(*
==============================================================================
 Method: EstimateTotalTime
------------------------------------------------------------------------------
 Purpose:
   - Estimate the total duration (in seconds) of the prime phase for the
     current recipe, based on how many different solvents (1..4) are used.
   - This is used solely for the HMI progress bar to give a rough visual
     indication of progress.

 Logic:
   1) Build a local array bLocalPrimeRequired[1..4] from the recipe, similar
      to BuildPrimeListFromRecipe.
   2) Count how many solvents are required (iCount).
   3) If iCount = 0 → return a small non-zero time (1.0 s) to avoid div by 0.
   4) Else → estimate = rTimePerSolvent * iCount * 7
      (the factor 7 is an empirical scaling based on test runs).
==============================================================================
*)
METHOD EstimateTotalTime : REAL
VAR
    iStage              : INT;
    iSolventNum         : INT;
    bLocalPrimeRequired : ARRAY[1..4] OF BOOL := [FALSE, FALSE, FALSE, FALSE];
    iCount              : INT := 0;
    rTimePerSolvent     : REAL := 15.0;   // Approximate time (s) to prime one solvent
END_VAR
// Build a local "prime required" list based on the active recipe
FOR iStage := 1 TO 4 DO
    iSolventNum := GVL_Recipe.stActiveRecipe.stSolventsTimes.aSolventN[iStage];

    IF (iSolventNum >= 1) AND (iSolventNum <= 4) THEN
        bLocalPrimeRequired[iSolventNum] := TRUE;
    END_IF
END_FOR

// Count how many solvents need priming
FOR iStage := 1 TO 4 DO
    IF bLocalPrimeRequired[iStage] THEN
        iCount := iCount + 1;
    END_IF
END_FOR

// If nothing to prime, return a small value to avoid division by zero
IF iCount = 0 THEN
    EstimateTotalTime := 1.0;
ELSE
    EstimateTotalTime := rTimePerSolvent * TO_REAL(iCount) * 7.0;
END_IF
END_METHOD

ACTION PrimeSolventCycle:
(*
==============================================================================
 PrimeSolventCycle
------------------------------------------------------------------------------
 Purpose:
   - Execute the generic prime cycle for the solvent indicated by
     iActiveSolventPosition (1..4).
   - This action uses iStepCounter as an internal step machine and sets
     bMovementComplete := TRUE when the cycle for the current solvent
     is finished.

 Prime sequence (per solvent):
   0) Initialise flags and HMI text for current solvent.
   1) Set valves [1..5] to the solvent position (1..4).
   2) Compute pump forward distances for rPrimeForwardVolume (ml).
   3) Pump forward (positive Distance) to pull solvent from bottle
      through the lines and into jars.
   4) Set valves [1..5] to needles position (6).
   5) Compute pump backward distances for rPrimeBackwardVolume (ml).
   6) Pump backward (negative Distance) to empty jars while keeping
      the lines filled with solvent.
   7) Set bMovementComplete := TRUE (cycle finished).
==============================================================================
*)

CASE iStepCounter OF

    // -------------------------------------------------------------
    // 0) Initialise HMI state and clear flags
    // -------------------------------------------------------------
    0:
        CASE iActiveSolventPosition OF
            1: GVL_HMI.HMIAnimation.sLoadTextRecovery := 'Prime Solvent 1';
            2: GVL_HMI.HMIAnimation.sLoadTextRecovery := 'Prime Solvent 2';
            3: GVL_HMI.HMIAnimation.sLoadTextRecovery := 'Prime Solvent 3';
            4: GVL_HMI.HMIAnimation.sLoadTextRecovery := 'Prime Solvent 4';
        ELSE
            GVL_HMI.HMIAnimation.sLoadTextRecovery := 'Prime Solvent';
        END_CASE;

        // Reset valve flags
        FOR i := 1 TO 5 DO
            bMoveValveDone[i] := FALSE;
        END_FOR

        // Reset pump flags and distances
        FOR i := 1 TO 10 DO
            bMovePumpDone[i] := FALSE;
            fDistance[i]     := 0.0;
        END_FOR

        bMovementComplete := FALSE;
        iStepCounter      := 1;


    // -------------------------------------------------------------
    // 1) Set valves [1..5] to the solvent position (1..4)
    // -------------------------------------------------------------
    1:
        FOR i := 1 TO 5 DO
            IF NOT bMoveValveDone[i] THEN
                bMoveValveDone[i] := GVL_Motion.aValvesObj[i].MoveValve(
                    iPosition := iActiveSolventPosition,   // solvent position 1..4
                    rVelocity := GVL_Motion.aValves[i].rTargetVel,
                    rAcc      := GVL_Motion.aValves[i].rAcceleration,
                    rDec      := GVL_Motion.aValves[i].rDeceleration
                );
            END_IF
        END_FOR

        // Wait until all valves reach solvent position
        IF bMoveValveDone[1] AND bMoveValveDone[2] AND bMoveValveDone[3]
           AND bMoveValveDone[4] AND bMoveValveDone[5] THEN

            FOR i := 1 TO 5 DO
                bMoveValveDone[i] := FALSE;
            END_FOR

            iStepCounter := 2;
        END_IF


    // -------------------------------------------------------------
    // 2) Calculate forward distance for rPrimeForwardVolume
    // -------------------------------------------------------------
    2:
        FOR i := 1 TO 10 DO
            fDistance[i] := F_VolumeToSteps(
                rVolume    := rPrimeForwardVolume,   // Forward prime volume
                iPumpIndex := i
            );
            bMovePumpDone[i] := FALSE;
        END_FOR

        iStepCounter := 3;


    // -------------------------------------------------------------
    // 3) Pump forward (positive movement) to fill lines and jars
    // -------------------------------------------------------------
    3:
        FOR i := 1 TO 10 DO
            IF NOT bMovePumpDone[i] THEN
                bMovePumpDone[i] := GVL_Motion.aPumpsRotary[i].MoveRelative(
                    Distance := fDistance[i],  // positive → forward
                    Velocity := GVL_Settings.stPumpParameters.iMeterVelocity * 6,
                    Acc      := GVL_Settings.stPumpParameters.iMeterVelocity * 3,
                    Dec      := GVL_Settings.stPumpParameters.iMeterVelocity * 3
                );
            END_IF
        END_FOR

        // Wait until all pumps finish forward prime
        IF bMovePumpDone[1] AND bMovePumpDone[2] AND bMovePumpDone[3] AND
           bMovePumpDone[4] AND bMovePumpDone[5] AND bMovePumpDone[6] AND
           bMovePumpDone[7] AND bMovePumpDone[8] AND bMovePumpDone[9] AND
           bMovePumpDone[10] THEN

            FOR i := 1 TO 10 DO
                bMovePumpDone[i] := FALSE;
            END_FOR

            iStepCounter := 4;
        END_IF


    // -------------------------------------------------------------
    // 4) Set valves [1..5] to needles position (6)
    // -------------------------------------------------------------
    4:
        FOR i := 1 TO 5 DO
            IF NOT bMoveValveDone[i] THEN
                bMoveValveDone[i] := GVL_Motion.aValvesObj[i].MoveValve(
                    iPosition := 6,   // needles position
                    rVelocity := GVL_Motion.aValves[i].rTargetVel,
                    rAcc      := GVL_Motion.aValves[i].rAcceleration,
                    rDec      := GVL_Motion.aValves[i].rDeceleration
                );
            END_IF
        END_FOR

        // Wait until all valves are at needles position
        IF bMoveValveDone[1] AND bMoveValveDone[2] AND bMoveValveDone[3]
           AND bMoveValveDone[4] AND bMoveValveDone[5] THEN

            FOR i := 1 TO 5 DO
                bMoveValveDone[i] := FALSE;
            END_FOR

            iStepCounter := 5;
        END_IF


    // -------------------------------------------------------------
    // 5) Calculate backward distance for rPrimeBackwardVolume
    // -------------------------------------------------------------
    5:
        FOR i := 1 TO 10 DO
            fDistance[i] := F_VolumeToSteps(
                rVolume    := rPrimeBackwardVolume,  // Backward prime volume
                iPumpIndex := i
            );
            bMovePumpDone[i] := FALSE;
        END_FOR

        iStepCounter := 6;


    // -------------------------------------------------------------
    // 6) Pump backward (negative movement) to empty jars into waste
    // -------------------------------------------------------------
    6:
        FOR i := 1 TO 10 DO
            IF NOT bMovePumpDone[i] THEN
                bMovePumpDone[i] := GVL_Motion.aPumpsRotary[i].MoveRelative(
                    Distance := -fDistance[i],  // negative → backward
                    Velocity := GVL_Settings.stPumpParameters.iRunVelocity * 6,
                    Acc      := GVL_Settings.stPumpParameters.iRunVelocity * 3,
                    Dec      := GVL_Settings.stPumpParameters.iRunVelocity * 3
                );
            END_IF
        END_FOR

        // Wait until all pumps finish backward cycle
        IF bMovePumpDone[1] AND bMovePumpDone[2] AND bMovePumpDone[3] AND
           bMovePumpDone[4] AND bMovePumpDone[5] AND bMovePumpDone[6] AND
           bMovePumpDone[7] AND bMovePumpDone[8] AND bMovePumpDone[9] AND
           bMovePumpDone[10] THEN

            FOR i := 1 TO 10 DO
                bMovePumpDone[i] := FALSE;
            END_FOR

            iStepCounter := 7;
        END_IF


    // -------------------------------------------------------------
    // 7) Prime cycle finished for this solvent
    // -------------------------------------------------------------
    7:
        bMovementComplete := TRUE;

END_CASE
END_ACTION

(*
==============================================================================
 Method: Reset
------------------------------------------------------------------------------
 Purpose:
   - Reset all internal flags, counters, and HMI fields associated with the
     prime phase, so that a new prime sequence can start cleanly.

 Behaviour:
   - Clears:
       * bStart, bBusy, bDone, bError, bProgressInitDone
       * ePrimeState, iStepCounter, bMovementComplete
       * bMoveValveDone[], bMovePumpDone[], fDistance[]
       * HMI prime text / bar (Recovery text cleared here as well)
   - Returns:
       Reset = TRUE once the operation is completed.
==============================================================================
*)
METHOD Reset : BOOL
VAR
    j : INT;
END_VAR
Reset := FALSE;

// Clear basic state and flags
bStart            := FALSE;
bBusy             := FALSE;
bDone             := FALSE;
bError            := FALSE;
bProgressInitDone := FALSE;

ePrimeState       := E_PrimeSolventState.PS_Idle;
iStepCounter      := 0;
bMovementComplete := FALSE;

// Clear motion flags and distances
FOR j := 1 TO 5 DO
    bMoveValveDone[j] := FALSE;
END_FOR

FOR j := 1 TO 10 DO
    bMovePumpDone[j] := FALSE;
    fDistance[j]     := 0.0;
END_FOR

// Clear HMI texts for prime / recovery bars if needed
GVL_HMI.HMIAnimation.sLoadTextRecovery := '';
GVL_HMI.HMIAnimation.rLoadBarRecovery  := 0.0;

// Mark reset as completed
Reset := TRUE;
RETURN;
END_METHOD

END_FUNCTION_BLOCK

// ---- POUs/Functions/F_AnyAxisMoving.TcPOU
FUNCTION F_AnyAxisMoving : BOOL
VAR_INPUT
END_VAR
VAR
	i : INT;
END_VAR

F_AnyAxisMoving := FALSE;

// Motors M1 - M3

F_AnyAxisMoving := F_AnyAxisMoving  OR (NOT GVL_Motion.M1Motor.iNotMoving)
									OR (NOT GVL_Motion.M2Motor.iNotMoving)
									OR (NOT GVL_Motion.M3Motor.iNotMoving);

// VICI Valves
FOR i := 1 TO 5 DO
    F_AnyAxisMoving := F_AnyAxisMoving 
        OR (NOT GVL_Motion.aValves[i].iNotMoving);
END_FOR

// Linear pumps
FOR i := 1 TO 10 DO
    F_AnyAxisMoving := F_AnyAxisMoving 
        OR (NOT GVL_Motion.aPumps[i].Linear.iNotMoving);
END_FOR

// Rotary pumps
FOR i := 1 TO 10 DO
    F_AnyAxisMoving := F_AnyAxisMoving 
        OR (NOT GVL_Motion.aPumps[i].Rotary.iNotMoving);
END_FOR

END_FUNCTION

// ---- POUs/1. MachineControl/PRG_SystemInit.TcPOU
PROGRAM PRG_SystemInit
VAR_OUTPUT
	bDone           : BOOL := FALSE;
END_VAR
VAR
	i               : INT;
	j				: INT;
    bAllDone        : BOOL := FALSE;
    bStartedAction  : BOOL := FALSE;
	bMoveZeroDone	: BOOL := FALSE;
    bInitComplete   : BOOL := FALSE;
	bVerticalMotorsDone		: BOOL := FALSE;   
	bLinearMotorsHomingDone	: BOOL := FALSE; 
	bValvesHomingDone 		: BOOL := FALSE;
	bLinearPumpsDone		: BOOL := FALSE;
	bPerformHoming			: BOOL := FALSE;
	
	bAllResetDone		: BOOL := FALSE;
	bEnableDone			: BOOL := FALSE;
	bResetCheck			: ARRAY[1..28] OF BOOL;
	
	aMotorsEnabled 	: ARRAY[1..3] OF BOOL;
	aValvesEnabled 	: ARRAY[1..5] OF BOOL;
	aLinearPumpsEnabled	: ARRAY[1..10] OF BOOL;
	aRotaryPumpsEnabled	: ARRAY[1..10] OF BOOL;
	
	bAllPumpsEnabled  : BOOL := FALSE;
	bAllLinearPumpsEnabled  : BOOL := FALSE;
	bAllRotaryPumpsEnabled  : BOOL := FALSE;
	bAllMotorsEnabled : BOOL := FALSE;
	bAllValvesEnabled : BOOL := FALSE;
	
	bHomeMotorDone	: ARRAY[1..3] OF BOOL;
	bHomeValveDone  : ARRAY[1..5] OF BOOL;
	bHomePumpDone	: ARRAY[1..10] OF BOOL;
	
	bM2InPosition	: BOOL;
	rPosTolerance	: REAL := 1.0;
	
	bMoveValve1Request	: BOOL := TRUE;
	bMoveValve2Request	: BOOL := TRUE;
	
	bMoveMotorsRequest	: ARRAY[1..3] OF BOOL;
	bMoveMotorDone		: ARRAY[1..3] OF BOOL;
	
	bCalibrationReset	  : BOOL := FALSE;
	bManualModeReset	  : BOOL := FALSE;
	bAutoCycleReset		  : BOOL := FALSE;
	bAllLogicResetDone	  : BOOL := FALSE;
	bInitLogicLatchesDone : BOOL := FALSE;
	
	tonResetDelay	: ton;
	tonEnableDelay	: ton;
	
	//Timeout timers for each step
	tonResetTimeOut		: ton;
	tonEnableTimeOut	: ton;
	tonHomeTimeOut		: ton;
	tonMoveAbsTimeOut	: ton;
		
	stStatus : ST_ActuatorStatus;
	
END_VAR

// ============================================================================
// PRG_SystemInit
// Handles full system initialization sequence:
//  0) Reset PRG's Manual | Calibration | AutoCycle
//  1) Reset all axes (motors, valves, pumps)
//  2) Enable all required axes
//  3) Perform homing on first startup OR move axes to zero on subsequent inits
//  4) Check completion and errors
//  5) Set bDone when initialization is complete
// ============================================================================

// ---------------------------------------------------------------------------
// 0) Basic delays between phases
// ---------------------------------------------------------------------------

// Delay before starting Reset
tonResetDelay(
    IN := NOT bAllResetDone,
    PT := T#1S
);

// Delay before starting Enable (only after Reset is fully done)
tonEnableDelay(
    IN := bAllResetDone AND NOT bEnableDone,
    PT := T#1S
);

// ---------------------------------------------------------------------------
// 0) Step 0 - Reset all logic Flags, PRGs and FBs
// ---------------------------------------------------------------------------
IF NOT bInitLogicLatchesDone AND GVL_Motion.bValvesPositionRecovered THEN ACT_ResetCommandFlags(); END_IF // Valves position recovery after shutdown change | Renan 22Jan2026

IF NOT bAllLogicResetDone AND bInitLogicLatchesDone THEN ACT_LogicResets(); END_IF

// ---------------------------------------------------------------------------
// 1) Step 1 - Reset all axes (motors, valves, linear and rotary pumps)
// ---------------------------------------------------------------------------
IF NOT bAllResetDone AND bAllLogicResetDone AND bInitLogicLatchesDone AND tonResetDelay.Q THEN
    ACT_ResetMotors();   // Uses bResetCheck[1..28], tonResetTimeOut, etc.
END_IF

// ---------------------------------------------------------------------------
// 2) Step 2 - Enable all axes (motors, valves, rotary pumps)
//     - Uses extra layer: checks Axis.Status.Error before/after Enable
// ---------------------------------------------------------------------------
IF bAllResetDone AND NOT bEnableDone AND tonEnableDelay.Q THEN
    ACT_EnableMotors();
END_IF

// ---------------------------------------------------------------------------
// 3) Step 3 - Decide if we need Homing or only MoveToZero
//     - First SystemInit: perform homing (bInitialHomingDone = FALSE)
//     - Next SystemInits: only move motors/valves to zero/home position
// ---------------------------------------------------------------------------

IF NOT bStartedAction AND bAllResetDone AND bEnableDone THEN
    bStartedAction := TRUE;

    // First time the machine starts: perform initial homing
    IF NOT GVL_Motion.bInitialHomingDone THEN
        bPerformHoming := TRUE;   // ACT_Homing() will be called
    ELSE
        bPerformHoming := FALSE;  // ACT_MoveToZero() will be called
    END_IF
END_IF

// ---------------------------------------------------------------------------
// 3a) Execute Homing or MoveToZero depending on bPerformHoming
// ---------------------------------------------------------------------------
IF bStartedAction THEN
    IF bPerformHoming THEN
        ACT_Homing();
    ELSE
        ACT_MoveToZero();
    END_IF
END_IF

// ---------------------------------------------------------------------------
// 4) Step 4 + 5 - Check if all motors and valves have completed their action
//     - Also checks for errors from wrapper (stStatus.bError)
//       and directly from Axis.Status.Error
// ---------------------------------------------------------------------------
IF bStartedAction AND bMoveZeroDone THEN
    bAllDone := TRUE;

    // Check motors M1..M3
    FOR i := 1 TO 3 DO
        stStatus := GVL_Motion.aMotors[i].GetStatus();

        // If any motor is not done yet
        IF NOT stStatus.bDone THEN
            bAllDone := FALSE;
        END_IF

        // If any motor returned an error (wrapper OR Axis), abort with immediate fault
        IF stStatus.bError THEN
            GVL_HMI.eMachineMode := E_MachineMode.IMEDIATE_FAULT;
            RETURN;
        END_IF
    END_FOR

    // Check valves V1..V5
    FOR i := 1 TO 5 DO
        stStatus := GVL_Motion.aValvesObj[i].GetStatus();

        // If any valve is not done yet
        IF NOT stStatus.bDone THEN
            bAllDone := FALSE;
        END_IF

        // If any valve returned an error (wrapper OR Axis), abort with immediate fault
        IF stStatus.bError THEN
            GVL_HMI.eMachineMode := E_MachineMode.IMEDIATE_FAULT;
            RETURN;
        END_IF
    END_FOR
END_IF

// ---------------------------------------------------------------------------
// 5) Step 6 - Finalization of System Init
//     - Set bDone only when Reset, Enable and Actions are all completed
// ---------------------------------------------------------------------------
IF bAllDone AND bAllResetDone AND bEnableDone AND NOT bInitComplete THEN
    bInitComplete := TRUE;
    bDone         := TRUE;

    // Mark that the initial homing has been successfully completed
    IF NOT GVL_Motion.bInitialHomingDone THEN
        GVL_Motion.bInitialHomingDone := TRUE;
    END_IF
END_IF

ACTION ACT_EnableMotors:
// ============================================================================
// Step 2: Enable all motors, valves and rotary pumps
//   - Uses aMotorsEnabled[1..3], aValvesEnabled[1..5], aRotaryPumpsEnabled[1..10]
//   - Sets bAllMotorsEnabled, bAllValvesEnabled, bAllRotaryPumpsEnabled
//   - Uses tonEnableTimeOut and GVL_Alarms.sMotionEnableTimeoutAxis
//   - Extra layer: checks wrapper error (GetStatus().bError) before enabling
// ============================================================================

IF NOT bEnableDone THEN

    // Assume all will be enabled, then AND with each device
    bAllMotorsEnabled      := TRUE;
    bAllValvesEnabled      := TRUE;
    bAllRotaryPumpsEnabled := TRUE;

    // -----------------------------
    // 2.1 Motors (M1..M3)
    // -----------------------------
    FOR i := 1 TO 3 DO
        // Read wrapper status
        stStatus := GVL_Motion.aMotors[i].GetStatus();

        // If wrapper reports error at this stage, abort System Init
        IF stStatus.bError THEN
            GVL_HMI.eMachineMode := E_MachineMode.IMEDIATE_FAULT;
            RETURN;
        END_IF

        // If axis is disabled, request Enable through wrapper
        // (If your wrapper has a specific bEnabled flag, you can check it here.
        // Otherwise, just call Enable() and rely on the wrapper to handle it.)
        aMotorsEnabled[i] := GVL_Motion.aMotors[i].Enable();

        bAllMotorsEnabled := bAllMotorsEnabled AND aMotorsEnabled[i];
    END_FOR

    // -----------------------------
    // 2.2 Valves (V1..V5)
    // -----------------------------
    FOR i := 1 TO 5 DO
        stStatus := GVL_Motion.aValvesObj[i].GetStatus();

        IF stStatus.bError THEN
            GVL_HMI.eMachineMode := E_MachineMode.IMEDIATE_FAULT;
            RETURN;
        END_IF

        aValvesEnabled[i] := GVL_Motion.aValvesObj[i].Enable();

        bAllValvesEnabled := bAllValvesEnabled AND aValvesEnabled[i];
    END_FOR

    // -----------------------------
    // 2.3 Rotary pumps (RP1..RP10)
// -----------------------------
    FOR i := 1 TO 10 DO
        stStatus := GVL_Motion.aPumpsRotary[i].GetStatus();

        IF stStatus.bError THEN
            GVL_HMI.eMachineMode := E_MachineMode.IMEDIATE_FAULT;
            RETURN;
        END_IF

        aRotaryPumpsEnabled[i] := GVL_Motion.aPumpsRotary[i].Enable();

        bAllRotaryPumpsEnabled := bAllRotaryPumpsEnabled AND aRotaryPumpsEnabled[i];
    END_FOR

    // -----------------------------
    // 2.4 Enable timeout monitoring and alarm
    // -----------------------------
    tonEnableTimeOut(IN := TRUE, PT := T#10S);

    IF tonEnableTimeOut.Q AND NOT (bAllMotorsEnabled AND bAllValvesEnabled AND bAllRotaryPumpsEnabled) THEN
        // Build string with axes that were NOT enabled within timeout

        // Motors M1..M3
        FOR i := 1 TO 3 DO
            IF NOT aMotorsEnabled[i] THEN
                IF GVL_Alarms.sMotionEnableTimeoutAxis <> '' THEN
                    GVL_Alarms.sMotionEnableTimeoutAxis :=
                        CONCAT(GVL_Alarms.sMotionEnableTimeoutAxis, ', ');
                END_IF
                GVL_Alarms.sMotionEnableTimeoutAxis :=
                    CONCAT(GVL_Alarms.sMotionEnableTimeoutAxis,
                           GVL_Constant.sMotionText[i]);
            END_IF
        END_FOR

        // Valves V1..V5
        FOR i := 1 TO 5 DO
            IF NOT aValvesEnabled[i] THEN
                IF GVL_Alarms.sMotionEnableTimeoutAxis <> '' THEN
                    GVL_Alarms.sMotionEnableTimeoutAxis :=
                        CONCAT(GVL_Alarms.sMotionEnableTimeoutAxis, ', ');
                END_IF
                GVL_Alarms.sMotionEnableTimeoutAxis :=
                    CONCAT(GVL_Alarms.sMotionEnableTimeoutAxis,
                           GVL_Constant.sMotionText[i + 3]);
            END_IF
        END_FOR

        // Rotary pumps RP1..RP10
        FOR i := 1 TO 10 DO
            IF NOT aRotaryPumpsEnabled[i] THEN
                IF GVL_Alarms.sMotionEnableTimeoutAxis <> '' THEN
                    GVL_Alarms.sMotionEnableTimeoutAxis :=
                        CONCAT(GVL_Alarms.sMotionEnableTimeoutAxis, ', ');
                END_IF
                GVL_Alarms.sMotionEnableTimeoutAxis :=
                    CONCAT(GVL_Alarms.sMotionEnableTimeoutAxis,
                           GVL_Constant.sMotionText[i + 18]);
            END_IF
        END_FOR

        GVL_Alarms.bMotionEnableTimeout := TRUE;
        // Strong robustness: abort System Init on enable timeout
        GVL_HMI.eMachineMode := E_MachineMode.IMEDIATE_FAULT;
        RETURN;
    END_IF

    // -----------------------------
    // 2.5 Step completion
    // -----------------------------
    IF bAllMotorsEnabled AND bAllValvesEnabled AND bAllRotaryPumpsEnabled THEN
        bEnableDone := TRUE;
        tonEnableTimeOut(IN := FALSE);
    END_IF

ELSE
    // Already done, ensure timer is off
    tonEnableTimeOut(IN := FALSE);
END_IF
END_ACTION

ACTION ACT_Homing:
// ============================================================================
// Step 3 (part 1): Initial homing sequence
//   - Only used when GVL_Motion.bInitialHomingDone = FALSE
//   - Homes vertical motors, then horizontal motor
//   - Moves valves to home position (position 5) when positions are recovered
//   - Monitors homing timeout and raises alarm
// ============================================================================

IF bPerformHoming THEN

    // -----------------------------
    // 3.1 Vertical motors homing (M1, M2)
    // -----------------------------
    IF NOT bHomeMotorDone[1] THEN
        bHomeMotorDone[1] := GVL_Motion.aMotors[1].Home(
            pHomeSensor := ADR(GVL_IO.gDigInputs.bStageCollection_Home),
            rVelocity   := GVL_Motion.M1Motor.rHomeVel,
            rAcc        := GVL_Motion.M1Motor.rHomeAcc,
            rDec        := GVL_Motion.M1Motor.rHomeDec
        );
    END_IF

    IF NOT bHomeMotorDone[2] THEN
        bHomeMotorDone[2] := GVL_Motion.aMotors[2].Home(
            pHomeSensor := ADR(GVL_IO.gDigInputs.bSampleRecovery_Vertical_Home),
            rVelocity   := GVL_Motion.M2Motor.rHomeVel,
            rAcc        := GVL_Motion.M2Motor.rHomeAcc,
            rDec        := GVL_Motion.M2Motor.rHomeDec
        );
    END_IF

    // Check if vertical motors homing is done
    IF bHomeMotorDone[1] AND bHomeMotorDone[2] THEN
        bVerticalMotorsDone := TRUE;
    END_IF

    // -----------------------------
    // 3.2 Horizontal motor homing (M3), only after verticals are done
    // -----------------------------
    IF bVerticalMotorsDone AND NOT bHomeMotorDone[3] THEN
        bHomeMotorDone[3] := GVL_Motion.aMotors[3].Home(
            pHomeSensor := ADR(GVL_IO.gDigInputs.bSampleRecovery_Horizontal_Home),
            rVelocity   := GVL_Motion.M3Motor.rHomeVel,
            rAcc        := GVL_Motion.M3Motor.rHomeAcc,
            rDec        := GVL_Motion.M3Motor.rHomeDec
        );
    END_IF

    // Check if all linear motors are homed
    IF bHomeMotorDone[1] AND bHomeMotorDone[2] AND bHomeMotorDone[3] THEN
        bLinearMotorsHomingDone := TRUE;
    END_IF

    // -----------------------------
    // 3.3 Valves homing (move to position 5) if position is recovered
    // -----------------------------
    IF GVL_Motion.bValvesPositionRecovered THEN
        // Move all valves to position 5 (home position)
        IF NOT bHomeValveDone[1] THEN
            bHomeValveDone[1] := GVL_Motion.aValvesObj[1].MoveValve(
                iPosition := 5,
                rVelocity := GVL_Motion.aValves[1].rHomeVel,
                rAcc      := GVL_Motion.aValves[1].rHomeAcc,
                rDec      := GVL_Motion.aValves[1].rHomeDec
            );
        END_IF

        IF NOT bHomeValveDone[2] THEN
            bHomeValveDone[2] := GVL_Motion.aValvesObj[2].MoveValve(
                iPosition := 5,
                rVelocity := GVL_Motion.aValves[2].rHomeVel,
                rAcc      := GVL_Motion.aValves[2].rHomeAcc,
                rDec      := GVL_Motion.aValves[2].rHomeDec
            );
        END_IF

        IF NOT bHomeValveDone[3] THEN
            bHomeValveDone[3] := GVL_Motion.aValvesObj[3].MoveValve(
                iPosition := 5,
                rVelocity := GVL_Motion.aValves[3].rHomeVel,
                rAcc      := GVL_Motion.aValves[3].rHomeAcc,
                rDec      := GVL_Motion.aValves[3].rHomeDec
            );
        END_IF

        IF NOT bHomeValveDone[4] THEN
            bHomeValveDone[4] := GVL_Motion.aValvesObj[4].MoveValve(
                iPosition := 5,
                rVelocity := GVL_Motion.aValves[4].rHomeVel,
                rAcc      := GVL_Motion.aValves[4].rHomeAcc,
                rDec      := GVL_Motion.aValves[4].rHomeDec
            );
        END_IF

        IF NOT bHomeValveDone[5] THEN
            bHomeValveDone[5] := GVL_Motion.aValvesObj[5].MoveValve(
                iPosition := 5,
                rVelocity := GVL_Motion.aValves[5].rHomeVel,
                rAcc      := GVL_Motion.aValves[5].rHomeAcc,
                rDec      := GVL_Motion.aValves[5].rHomeDec
            );
        END_IF
    END_IF

    // Check if all valves homing are done
    bValvesHomingDone :=
        bHomeValveDone[1] AND bHomeValveDone[2] AND bHomeValveDone[3] AND
        bHomeValveDone[4] AND bHomeValveDone[5];

	// If all motors and valves completed their homing, finalize
	IF bLinearMotorsHomingDone AND bValvesHomingDone THEN 
		bMoveZeroDone := TRUE;
	END_IF	
	
    // -----------------------------
    // 3.4 Homing timeout monitoring and alarm
    // -----------------------------
    tonHomeTimeOut(
        IN := NOT (bLinearMotorsHomingDone AND bValvesHomingDone),
        PT := T#40S
    );

    IF tonHomeTimeOut.Q AND NOT (bLinearMotorsHomingDone AND bValvesHomingDone) THEN
        // Build string with axes that were NOT homed in time

        // Motors M1..M3
        FOR j := 1 TO 3 DO
            IF NOT bHomeMotorDone[j] THEN
                IF GVL_Alarms.sMotionHomeTimeoutAxis <> '' THEN
                    GVL_Alarms.sMotionHomeTimeoutAxis :=
                        CONCAT(GVL_Alarms.sMotionHomeTimeoutAxis, ', ');
                END_IF
                GVL_Alarms.sMotionHomeTimeoutAxis :=
                    CONCAT(GVL_Alarms.sMotionHomeTimeoutAxis,
                           GVL_Constant.sMotionText[j]);
            END_IF
        END_FOR

        // Valves V1..V5
        FOR j := 1 TO 5 DO
            IF NOT bHomeValveDone[j] THEN
                IF GVL_Alarms.sMotionHomeTimeoutAxis <> '' THEN
                    GVL_Alarms.sMotionHomeTimeoutAxis :=
                        CONCAT(GVL_Alarms.sMotionHomeTimeoutAxis, ', ');
                END_IF
                GVL_Alarms.sMotionHomeTimeoutAxis :=
                    CONCAT(GVL_Alarms.sMotionHomeTimeoutAxis,
                           GVL_Constant.sMotionText[j + 3]);
            END_IF
        END_FOR

        GVL_Alarms.bMotionHomeTimeout := TRUE;
        GVL_HMI.eMachineMode          := E_MachineMode.IMEDIATE_FAULT;
    END_IF

END_IF
END_ACTION

ACTION ACT_LogicResets:
IF NOT bAllLogicResetDone THEN
	
	bCalibrationReset	:= PRG_Calibration.Reset();
	bManualModeReset	:= PRG_ManualControl.Reset();
	bAutoCycleReset		:= PRG_AutoCycle.Reset();
	
	IF bCalibrationReset AND bManualModeReset AND bAutoCycleReset THEN
		bAllLogicResetDone 	:= TRUE;
	END_IF
	
END_IF
END_ACTION

ACTION ACT_MoveToZero:
// ============================================================================
// Step 3 (part 2): Move motors and valves to zero / default positions
//   - Used when GVL_Motion.bInitialHomingDone = TRUE
//   - Moves:
//       - M1, M2, M3 -> position 0.0
//       - Valves V1..V5 -> position 5
//   - Uses bMoveMotorDone[1..3] and bHomeValveDone[1..5]
//   - Monitors move absolute timeout and raises alarm
// ============================================================================

IF NOT bPerformHoming THEN

    // -----------------------------
    // 3.5 Move linear motors to 0.0
    // -----------------------------
    // You can adjust these velocity/acc/dec parameters as needed
    IF NOT bMoveMotorDone[1] THEN
        bMoveMotorDone[1] := GVL_Motion.aMotors[1].MoveAbsolute(
            rPosition := GVL_Settings.stMachineParam.aM1Position[1],
            rVelocity := GVL_Settings.stMachineParam.rM1Velocity,
            rAcc      := GVL_Settings.stMachineParam.rM1Accleration,
            rDec      := GVL_Settings.stMachineParam.rM1Deceleration
        );
    END_IF

    IF NOT bMoveMotorDone[2] THEN
        bMoveMotorDone[2] := GVL_Motion.aMotors[2].MoveAbsolute(
            rPosition := GVL_Settings.stMachineParam.aM2Position[1],
            rVelocity := GVL_Settings.stMachineParam.rM2Velocity,
            rAcc      := GVL_Settings.stMachineParam.rM2Accleration,
            rDec      := GVL_Settings.stMachineParam.rM2Deceleration
        );
    END_IF
	
	// Track real M2 Position before start moving M3 
	bM2InPosition := ABS(GVL_Motion.M2Motor.rActualPos - GVL_Settings.stMachineParam.aM2Position[1]) < rPosTolerance;
	
    IF bMoveMotorDone[2] AND bM2InPosition AND NOT bMoveMotorDone[3] THEN
        bMoveMotorDone[3] := GVL_Motion.aMotors[3].MoveAbsolute(
            rPosition := GVL_Settings.stMachineParam.aM3Position[1],
            rVelocity := GVL_Settings.stMachineParam.rM3Velocity,
            rAcc      := GVL_Settings.stMachineParam.rM3Accleration,
            rDec      := GVL_Settings.stMachineParam.rM3Deceleration
        );
    END_IF

    // Linear motors move done flag
    bLinearMotorsHomingDone :=
        bMoveMotorDone[1] AND bMoveMotorDone[2] AND bMoveMotorDone[3];

    // -----------------------------
    // 3.6 Move valves to position 5 (default/home position)
// -----------------------------
    IF NOT bHomeValveDone[1] THEN
        bHomeValveDone[1] := GVL_Motion.aValvesObj[1].MoveValve(
            iPosition := 5,
            rVelocity := GVL_Motion.aValves[1].rHomeVel,
            rAcc      := GVL_Motion.aValves[1].rHomeAcc,
            rDec      := GVL_Motion.aValves[1].rHomeDec
        );
    END_IF

    IF NOT bHomeValveDone[2] THEN
        bHomeValveDone[2] := GVL_Motion.aValvesObj[2].MoveValve(
            iPosition := 5,
            rVelocity := GVL_Motion.aValves[2].rHomeVel,
            rAcc      := GVL_Motion.aValves[2].rHomeAcc,
            rDec      := GVL_Motion.aValves[2].rHomeDec
        );
    END_IF

    IF NOT bHomeValveDone[3] THEN
        bHomeValveDone[3] := GVL_Motion.aValvesObj[3].MoveValve(
            iPosition := 5,
            rVelocity := GVL_Motion.aValves[3].rHomeVel,
            rAcc      := GVL_Motion.aValves[3].rHomeAcc,
            rDec      := GVL_Motion.aValves[3].rHomeDec
        );
    END_IF

    IF NOT bHomeValveDone[4] THEN
        bHomeValveDone[4] := GVL_Motion.aValvesObj[4].MoveValve(
            iPosition := 5,
            rVelocity := GVL_Motion.aValves[4].rHomeVel,
            rAcc      := GVL_Motion.aValves[4].rHomeAcc,
            rDec      := GVL_Motion.aValves[4].rHomeDec
        );
    END_IF

    IF NOT bHomeValveDone[5] THEN
        bHomeValveDone[5] := GVL_Motion.aValvesObj[5].MoveValve(
            iPosition := 5,
            rVelocity := GVL_Motion.aValves[5].rHomeVel,
            rAcc      := GVL_Motion.aValves[5].rHomeAcc,
            rDec      := GVL_Motion.aValves[5].rHomeDec
        );
    END_IF

    // Valves move done flag
    bValvesHomingDone :=
        bHomeValveDone[1] AND bHomeValveDone[2] AND
        bHomeValveDone[3] AND bHomeValveDone[4] AND bHomeValveDone[5];
	
	// If all motors and valves completed their homing, finalize
	IF bLinearMotorsHomingDone AND bValvesHomingDone THEN 
		bMoveZeroDone := TRUE;
	END_IF
	
    // -----------------------------
    // 3.7 MoveAbs timeout monitoring and alarm
    //    (Note: here we correctly use bMoveMotorDone instead of bHomeMotorDone)
// -----------------------------
    tonMoveAbsTimeOut(
        IN := NOT (bLinearMotorsHomingDone AND bValvesHomingDone),
        PT := T#40S
    );

    IF tonMoveAbsTimeOut.Q AND NOT (bLinearMotorsHomingDone AND bValvesHomingDone) THEN
        // Build string with axes that did NOT complete MoveAbsolute in time

        // Motors M1..M3
        FOR j := 1 TO 3 DO
            IF NOT bMoveMotorDone[j] THEN
                IF GVL_Alarms.sMotionMoveAbsTimeoutAxis <> '' THEN
                    GVL_Alarms.sMotionMoveAbsTimeoutAxis :=
                        CONCAT(GVL_Alarms.sMotionMoveAbsTimeoutAxis, ', ');
                END_IF
                GVL_Alarms.sMotionMoveAbsTimeoutAxis :=
                    CONCAT(GVL_Alarms.sMotionMoveAbsTimeoutAxis,
                           GVL_Constant.sMotionText[j]);
            END_IF
        END_FOR

        // Valves V1..V5
        FOR j := 1 TO 5 DO
            IF NOT bHomeValveDone[j] THEN
                IF GVL_Alarms.sMotionMoveAbsTimeoutAxis <> '' THEN
                    GVL_Alarms.sMotionMoveAbsTimeoutAxis :=
                        CONCAT(GVL_Alarms.sMotionMoveAbsTimeoutAxis, ', ');
                END_IF
                GVL_Alarms.sMotionMoveAbsTimeoutAxis :=
                    CONCAT(GVL_Alarms.sMotionMoveAbsTimeoutAxis,
                           GVL_Constant.sMotionText[j + 3]);
            END_IF
        END_FOR

        GVL_Alarms.bMotionMoveAbsTimeout := TRUE;
        GVL_HMI.eMachineMode             := E_MachineMode.IMEDIATE_FAULT;
    END_IF

END_IF
END_ACTION

ACTION ACT_ResetCommandFlags:
(*
    Action: ACT_ResetCommandFlags
    Purpose:
        Clear all HMI command flags and internal latched commands that might remain TRUE
        after an abnormal interruption (STOP/Abort), preventing unintended auto-start
        when re-entering a mode.

    Where to call:
        - PRG_StoppedState (first scan / when entering STOPPED)
        - PRG_SystemInit (first scan / at init start)

    Notes:
        - This action is safe to call repeatedly (idempotent).
        - Adjust array bounds if your project differs.
*)

// ============================================================
// 1) Calibration - HMI triggers (buttons / commands)
// ============================================================
GVL_HMI.bStartCalibrationBt        := FALSE;

GVL_HMI.bCalLeakTestButton         := FALSE;
GVL_HMI.bCalPressureUpSystemBt     := FALSE;
GVL_HMI.bCalHoldSysPressureBt      := FALSE;
GVL_HMI.bCalStopLeakTestBt         := FALSE;

GVL_HMI.bCalLinearPumpsEnableBt    := FALSE;
GVL_HMI.bCalLinearPumpsHomeBt      := FALSE;
GVL_HMI.bCalLinearPumpsMoveBt      := FALSE;
GVL_HMI.bCalLinearPumpsStopBt      := FALSE;
GVL_HMI.bCalLinearPumpsDirty       := FALSE;

GVL_HMI.bCalMoveValves             := FALSE;
GVL_HMI.bCalMoveM1Motor            := FALSE;

// Scale / CalBox popups / acknowledge flags
GVL_HMI.bScaleNeedsAtention        := FALSE;
GVL_HMI.bScaleFixed                := FALSE;
GVL_HMI.bCalBoxNeedsAttention      := FALSE;
GVL_HMI.bCalBoxFixed               := FALSE;


// ============================================================
// 2) Calibration - internal latches (must be cleared on STOP/Init)
// ============================================================
GVL_Calibration.bStartCalibration      := FALSE;
GVL_Calibration.bAbortCalibration      := FALSE;
GVL_Calibration.bStartCreationCalJson  := FALSE;
GVL_Calibration.bDosingTestEnable	   := FALSE;


// ============================================================
// 3) Manual Mode - motors / valves / pumps command arrays
// ============================================================

// Manual motors (adjust bounds if needed)
FOR i := 1 TO 3 DO
    GVL_HMI.aManualMotorsCmd[i].bRun  := FALSE;
    GVL_HMI.aManualMotorsCmd[i].bStop := FALSE;
END_FOR

// Manual valves
FOR i := 1 TO 5 DO
    GVL_HMI.aManualValvesCmd[i].bMove := FALSE;
    GVL_HMI.aManualValvesCmd[i].bStop := FALSE;
END_FOR

// Global pump buttons
GVL_HMI.bRunPumpsBySpeedBt  := FALSE;
GVL_HMI.bRunPumpsByVolumeBt := FALSE;

// Per-pump commands
FOR i := 1 TO 10 DO
    GVL_HMI.aManualPumpsCmd[i].bRunBySpeed  := FALSE;
    GVL_HMI.aManualPumpsCmd[i].bRunByVolume := FALSE;
    GVL_HMI.aManualPumpsCmd[i].bStop        := FALSE;
    GVL_HMI.aManualPumpsCmd[i].bActive      := FALSE;
END_FOR


// ============================================================
// 4) AutoCycle - popup/start/hold commands
// ============================================================
GVL_HMI.bShowAutoCyclePopup     	:= FALSE;
GVL_HMI.bStartAutoCycleButton   	:= FALSE;
GVL_HMI.bSystemReady_ReqAutoCycle 	:= FALSE;

GVL_HMI.bAutoCycleHoldReq       	:= FALSE;
GVL_HMI.bAutoCycleHoldActive    	:= FALSE;
GVL_HMI.bAutoCycleHoldPopup     	:= FALSE;
GVL_HMI.bAutoCycleContinueCmd   	:= FALSE;
GVL_HMI.bAutoCycleCancelCmd     	:= FALSE;


// ============================================================
// 5) Finishing
// ============================================================
bInitLogicLatchesDone := TRUE;
END_ACTION

ACTION ACT_ResetMotors:
// ============================================================================
// Step 1: Reset all motors, valves, linear and rotary pumps
// Uses array bResetCheck[1..28] to track each device:
//   1..3   -> Motors      (M1..M3)
//   4..8   -> Valves      (V1..V5)
//   9..18  -> Linear pumps  (LP1..LP10)
//   19..28 -> Rotary pumps  (RP1..RP10)
// ============================================================================

IF NOT bAllResetDone THEN

    // -----------------------------
    // 1.1 Motors (M1..M3)
    // -----------------------------
    IF NOT bResetCheck[1] THEN
        bResetCheck[1] := GVL_Motion.aMotors[1].Reset();
    END_IF

    IF NOT bResetCheck[2] THEN
        bResetCheck[2] := GVL_Motion.aMotors[2].Reset();
    END_IF

    IF NOT bResetCheck[3] THEN
        bResetCheck[3] := GVL_Motion.aMotors[3].Reset();
    END_IF

    // -----------------------------
    // 1.2 Valves (V1..V5)
    // -----------------------------
    IF NOT bResetCheck[4] THEN
        bResetCheck[4] := GVL_Motion.aValvesObj[1].Reset();
    END_IF

    IF NOT bResetCheck[5] THEN
        bResetCheck[5] := GVL_Motion.aValvesObj[2].Reset();
    END_IF

    IF NOT bResetCheck[6] THEN
        bResetCheck[6] := GVL_Motion.aValvesObj[3].Reset();
    END_IF

    IF NOT bResetCheck[7] THEN
        bResetCheck[7] := GVL_Motion.aValvesObj[4].Reset();
    END_IF

    IF NOT bResetCheck[8] THEN
        bResetCheck[8] := GVL_Motion.aValvesObj[5].Reset();
    END_IF

    // -----------------------------
    // 1.3 Linear pumps (LP1..LP10)
    // -----------------------------
    IF NOT bResetCheck[9] THEN
        bResetCheck[9] := GVL_Motion.aPumpsLinear[1].Reset();
    END_IF
    IF NOT bResetCheck[10] THEN
        bResetCheck[10] := GVL_Motion.aPumpsLinear[2].Reset();
    END_IF
    IF NOT bResetCheck[11] THEN
        bResetCheck[11] := GVL_Motion.aPumpsLinear[3].Reset();
    END_IF
    IF NOT bResetCheck[12] THEN
        bResetCheck[12] := GVL_Motion.aPumpsLinear[4].Reset();
    END_IF
    IF NOT bResetCheck[13] THEN
        bResetCheck[13] := GVL_Motion.aPumpsLinear[5].Reset();
    END_IF
    IF NOT bResetCheck[14] THEN
        bResetCheck[14] := GVL_Motion.aPumpsLinear[6].Reset();
    END_IF
    IF NOT bResetCheck[15] THEN
        bResetCheck[15] := GVL_Motion.aPumpsLinear[7].Reset();
    END_IF
    IF NOT bResetCheck[16] THEN
        bResetCheck[16] := GVL_Motion.aPumpsLinear[8].Reset();
    END_IF
    IF NOT bResetCheck[17] THEN
        bResetCheck[17] := GVL_Motion.aPumpsLinear[9].Reset();
    END_IF
    IF NOT bResetCheck[18] THEN
        bResetCheck[18] := GVL_Motion.aPumpsLinear[10].Reset();
    END_IF

    // -----------------------------
    // 1.4 Rotary pumps (RP1..RP10)
    // -----------------------------
    IF NOT bResetCheck[19] THEN
        bResetCheck[19] := GVL_Motion.aPumpsRotary[1].Reset();
    END_IF
    IF NOT bResetCheck[20] THEN
        bResetCheck[20] := GVL_Motion.aPumpsRotary[2].Reset();
    END_IF
    IF NOT bResetCheck[21] THEN
        bResetCheck[21] := GVL_Motion.aPumpsRotary[3].Reset();
    END_IF
    IF NOT bResetCheck[22] THEN
        bResetCheck[22] := GVL_Motion.aPumpsRotary[4].Reset();
    END_IF
    IF NOT bResetCheck[23] THEN
        bResetCheck[23] := GVL_Motion.aPumpsRotary[5].Reset();
    END_IF
    IF NOT bResetCheck[24] THEN
        bResetCheck[24] := GVL_Motion.aPumpsRotary[6].Reset();
    END_IF
    IF NOT bResetCheck[25] THEN
        bResetCheck[25] := GVL_Motion.aPumpsRotary[7].Reset();
    END_IF
    IF NOT bResetCheck[26] THEN
        bResetCheck[26] := GVL_Motion.aPumpsRotary[8].Reset();
    END_IF
    IF NOT bResetCheck[27] THEN
        bResetCheck[27] := GVL_Motion.aPumpsRotary[9].Reset();
    END_IF
    IF NOT bResetCheck[28] THEN
        bResetCheck[28] := GVL_Motion.aPumpsRotary[10].Reset();
    END_IF

    // -----------------------------------------------------------------------
    // 1.5 Check if all resets are done
    // -----------------------------------------------------------------------
    IF bResetCheck[1] AND bResetCheck[2] AND bResetCheck[3] AND
       bResetCheck[4] AND bResetCheck[5] AND bResetCheck[6] AND
       bResetCheck[7] AND bResetCheck[8] AND
       bResetCheck[9] AND bResetCheck[10] AND bResetCheck[11] AND
       bResetCheck[12] AND bResetCheck[13] AND bResetCheck[14] AND
       bResetCheck[15] AND bResetCheck[16] AND bResetCheck[17] AND
       bResetCheck[18] AND
       bResetCheck[19] AND bResetCheck[20] AND bResetCheck[21] AND
       bResetCheck[22] AND bResetCheck[23] AND bResetCheck[24] AND
       bResetCheck[25] AND bResetCheck[26] AND bResetCheck[27] AND
       bResetCheck[28] THEN
        bAllResetDone := TRUE;
    ELSE
        bAllResetDone := FALSE;
    END_IF

    // -----------------------------------------------------------------------
    // 1.6 Reset timeout monitoring and alarm trigger
    // -----------------------------------------------------------------------
    tonResetTimeOut(IN := TRUE, PT := T#10S);

    IF tonResetTimeOut.Q THEN
        // Build string with axes that were NOT reset within timeout
        FOR j := 1 TO 28 DO
            IF NOT bResetCheck[j] THEN
                IF GVL_Alarms.sMotionResetTimeoutAxis <> '' THEN
                    GVL_Alarms.sMotionResetTimeoutAxis :=
                        CONCAT(GVL_Alarms.sMotionResetTimeoutAxis, ', ');
                END_IF
                GVL_Alarms.sMotionResetTimeoutAxis :=
                    CONCAT(GVL_Alarms.sMotionResetTimeoutAxis,
                           GVL_Constant.sMotionText[j]);
            END_IF
        END_FOR

        GVL_Alarms.bMotionResetTimeout := TRUE;
        // Optional: you could also force IMEDIATE_FAULT here if desired
    END_IF

ELSE
    // Reset already completed, ensure timeout timer is off
    tonResetTimeOut(IN := FALSE);
END_IF
END_ACTION

METHOD Reset : BOOL
VAR_INPUT	
END_VAR
VAR
	i : INT;
END_VAR
// ============================================================================
// PRG_SystemInit.Reset()
// ---------------------------------------------------------------------------
// This method clears all internal flags, arrays and timers used by
// PRG_SystemInit so that a new initialization sequence can start from a
// clean state.
//
// Return:
//   TRUE  - Always returns TRUE after the internal context is fully reset.
//           (The actual System Init progress is controlled by bAllResetDone,
//            bEnableDone, bAllDone, etc. in the main body.)
//
// Typical usage (in PRG_MasterControl):
//   - When entering E_MachineMode.SYSTEM_INITIALIZING,
//     call PRG_SystemInit.Reset() once to clear the context.
// ============================================================================

Reset := FALSE; // Default return

// ---------------------------------------------------------------------------
// 1) Global step control flags
// ---------------------------------------------------------------------------
bAllResetDone           := FALSE;
bEnableDone             := FALSE;
bStartedAction          := FALSE;
bPerformHoming          := FALSE;
bInitComplete           := FALSE;
bAllDone                := FALSE;
bMoveZeroDone 			:= FALSE;
bM2InPosition			:= FALSE;
bDone                   := FALSE;   

bVerticalMotorsDone     := FALSE;
bLinearMotorsHomingDone := FALSE;
bValvesHomingDone       := FALSE;

bCalibrationReset 		:= FALSE;
bManualModeReset 		:= FALSE;
bAutoCycleReset	 		:= FALSE;
bAllLogicResetDone 		:= FALSE;
bInitLogicLatchesDone	:= FALSE;

// ---------------------------------------------------------------------------
// 2) Per-device reset tracking array (1..28)
//    1..3   -> Motors       (M1..M3)
//    4..8   -> Valves       (V1..V5)
//    9..18  -> Linear pumps (LP1..LP10)
//    19..28 -> Rotary pumps (RP1..RP10)
// ---------------------------------------------------------------------------
FOR i := 1 TO 28 DO
    bResetCheck[i] := FALSE;
END_FOR

// ---------------------------------------------------------------------------
// 3) Enable state arrays
//    Motors:        aMotorsEnabled[1..3]
//    Valves:        aValvesEnabled[1..5]
//    Rotary pumps:  aRotaryPumpsEnabled[1..10]
// ---------------------------------------------------------------------------
FOR i := 1 TO 3 DO
    aMotorsEnabled[i] := FALSE;
END_FOR

FOR i := 1 TO 5 DO
    aValvesEnabled[i] := FALSE;
END_FOR

FOR i := 1 TO 10 DO
    aRotaryPumpsEnabled[i] := FALSE;
END_FOR

bAllMotorsEnabled      := FALSE;
bAllValvesEnabled      := FALSE;
bAllRotaryPumpsEnabled := FALSE;

// ---------------------------------------------------------------------------
// 4) Homing / MoveToZero flags
//    - bHomeMotorDone[1..3] : homing done flags for M1..M3
//    - bMoveMotorDone[1..3] : move-to-zero done flags for M1..M3
//    - bHomeValveDone[1..5] : homing/move done flags for V1..V5
// ---------------------------------------------------------------------------
FOR i := 1 TO 3 DO
    bHomeMotorDone[i] := FALSE;
    bMoveMotorDone[i] := FALSE;
END_FOR

FOR i := 1 TO 5 DO
    bHomeValveDone[i] := FALSE;
END_FOR

// ---------------------------------------------------------------------------
// 5) Timers used in System Init
// ---------------------------------------------------------------------------

// Phase delays
tonResetDelay(IN := FALSE);
tonEnableDelay(IN := FALSE);

// Timeouts
tonResetTimeOut(IN := FALSE);
tonEnableTimeOut(IN := FALSE);
tonHomeTimeOut(IN := FALSE);
tonMoveAbsTimeOut(IN := FALSE);

// ---------------------------------------------------------------------------
// 6) Alarm strings and flags used by System Init
// ---------------------------------------------------------------------------

// Reset timeout
GVL_Alarms.sMotionResetTimeoutAxis := '';
GVL_Alarms.bMotionResetTimeout     := FALSE;

// Enable timeout
GVL_Alarms.sMotionEnableTimeoutAxis := '';
GVL_Alarms.bMotionEnableTimeout     := FALSE;

// Homing timeout
GVL_Alarms.sMotionHomeTimeoutAxis := '';
GVL_Alarms.bMotionHomeTimeout     := FALSE;

// Move Absolute timeout
GVL_Alarms.sMotionMoveAbsTimeoutAxis := '';
GVL_Alarms.bMotionMoveAbsTimeout     := FALSE;

// ---------------------------------------------------------------------------
// 7) Finalize
// ---------------------------------------------------------------------------
Reset := TRUE;
END_METHOD

END_PROGRAM

// ---- POUs/5. Calibration/PRG_Calibration.TcPOU
PROGRAM PRG_Calibration
VAR_OUTPUT
    bCalibrationFinished : BOOL;  // Done Flag
END_VAR
VAR
	fbLeakTest : FB_LeakTest;
	bLeakTestReset : BOOL := FALSE;
	
	bResetRequested : BOOL := FALSE;
	
	fbCalibrationManager : FB_CalibrationManager;
	fbSaveCalReport		 : FB_SaveCalibrationReport;

    bStartCalibrationPrev : BOOL;
    bStartCalibrationEdge : BOOL;
	
	iLastRepSetpoint : INT := -1;
	iDataCount : INT;
    i : INT;
	
	fbSolenoidControl	: FB_SolenoidControl;
	eStopState 			: E_StopState 		:= E_StopState.Init;
	ePState 			: E_PState 			:= E_PState.Init;	
	
	bPressureUpExecute 		: BOOL := FALSE;
    bPressureUpRequested 	: BOOL := FALSE;
	bSealStages				: BOOL := FALSE;
	bPressureUpSolenoids	: BOOL := FALSE;
	bHoldPressureExecute 	: BOOL := FALSE;
    bHoldPressureRequested 	: BOOL := FALSE;
	bHoldPressureSolenoids	: BOOL := FALSE;
	bStopLeakTestExecute 	: BOOL := FALSE;
    bStopLeakTestRequested 	: BOOL := FALSE;
	bStopLeakTestSolenoids 	: BOOL := FALSE;
	tonLeakTestStateDelay	: TON;
	
	iSelectedSolvent 		: USINT;
	rSelectedSolventDensity : LREAL;
	bValidSelectedSolvent 	: BOOL;
	
	bMoveIssued     : BOOL := FALSE;
	bNeedsSet 		: BOOL := FALSE;
    tonSealTimeout  : TON;
	
	bStopM1Motor 			: BOOL := FALSE;
	bResetM1Motor 			: BOOL := FALSE;
	tonResetMotorDelay 		: ton;
	
	bLinearPumpsEnabled		: BOOL := FALSE;
	bLinearPumpsHomed		: BOOL := FALSE;
	bLinearPumpsOldPosStart	: BOOL := FALSE;
	bLinearPumpsOldPosDone	: BOOL := FALSE;
	bLinearPumpsMove		: BOOL := FALSE;
	aLinearPumpsEnable 		: ARRAY[1..10] OF BOOL;
	aLinearPumpsDisable		: ARRAY[1..10] OF BOOL;
	aLinearPumpsHoming 		: ARRAY[1..10] OF BOOL;
	bLinearPumpsOldPosMove	: ARRAY[1..10] OF BOOL;
	aLinearPumpsMoveDone 	: ARRAY[1..10] OF BOOL; // Tracks per-axis move completion
	rtrigSaveLinearPumps	: R_TRIG;
	
	bCalPressureUpSystemBt: BOOL;
	
	//Valves movement
	bMoveValves	: ARRAY[1..5] OF BOOL;
	bMoveM1Fast	: BOOL := FALSE;
	bMoveM1Slow	: BOOL := FALSE;
	
	bResetDone	: BOOL := FALSE;
	
	// Temp Dosing Test
	bDosingTestEnable  : BOOL := FALSE;
	aDosingPumps	   : ARRAY[1..10] OF BOOL := [FALSE, FALSE, TRUE, FALSE, FALSE, FALSE, TRUE, FALSE, FALSE, FALSE];
	bSetDosingPumps	   : BOOL := FALSE;
	fbDosingTest	   : FB_DosingTest;
	bDosingTestReset   : BOOL := FALSE;
	bDosingTestResults  : BOOL := FALSE;
	iReplicates			: USINT := 3;
	rTargetVolume		: LREAL := 50.0;
	
END_VAR

DB_Create_Calibration();	//Create a new calibration inside the DB.

IF GVL_HMI.bCalLeakTestButton THEN
	bLeakTestReset := FALSE;
END_IF

(* Scale *) //------------------------------------------------------------------------------------------------------------------------------------------------------------
// Instancing and calling fbScaleDevice object
GVL_Calibration.fbScaleDevice(sRemoteHost := GVL_Settings.aBalanceIP, nRemotePort := GVL_Settings.nBalancePort);

(* Leak Test *) //--------------------------------------------------------------------------------------------------------------------------------------------------------
// Leak Test request from HMI
fbLeakTest(	bExecute := GVL_HMI.bCalLeakTestButton, 
			eSolenoidPosition := E_SolenoidSet.LEAKTEST, 
			tMonitorTime := GVL_Settings.stLeakTestParameters.tLeakTestMonitorTime, 
			tPressureUpTime := GVL_Settings.stLeakTestParameters.tLeakTestBuildUpTime 
			);

// Leak Test post treatment
IF fbLeakTest.bLeakTestDone AND NOT fbLeakTest.bLeakTestError THEN
	GVL_HMI.bCalLeakTestPass := TRUE;
	GVL_HMI.bCalLeakTestError := FALSE;
	GVL_HMI.bCalLeakTestButton := FALSE;
	IF NOT bLeakTestReset THEN
		bLeakTestReset := fbLeakTest.Reset();
	END_IF
END_IF

IF fbLeakTest.bLeakTestError THEN
	GVL_HMI.bCalLeakTestError := TRUE;
	GVL_HMI.bCalLeakTestPass := FALSE;
	GVL_HMI.bCalLeakTestButton := FALSE;
	IF NOT bLeakTestReset THEN
		bLeakTestReset := fbLeakTest.Reset();
	END_IF
END_IF

tonLeakTestStateDelay( IN := ((GVL_HMI.bCalLeakTestError OR GVL_HMI.bCalLeakTestPass) AND NOT GVL_HMI.bCalLeakTestButton), PT := T#10S);

IF tonLeakTestStateDelay.Q THEN
	GVL_HMI.sCalLeakTestStatus := 'Idle';
	GVL_HMI.iCalLeakTestState  := 1;
END_IF

// HMI Button responsible for pressurize the system
IF GVL_HMI.bCalPressureUpSystemBt THEN
	IF GVL_Settings.stMachineParam.aM1Position[2] >= (GVL_Motion.M1Motor.rActualPos - 5) THEN
		GVL_HMI.bCalPressureUpSystemBt := NOT GVL_IO.gSetSolenoidControl.PressureUp(); //PressureUp();
	ELSE
		//Raise interlock alarm
		GVL_HMI.bCalPressureUpSystemBt := FALSE;
	END_IF
END_IF

// HMI Button responsible for hold the air in the system after the system pressure up
IF GVL_HMI.bCalHoldSysPressureBt THEN
	IF GVL_Settings.stMachineParam.aM1Position[2] >= (GVL_Motion.M1Motor.rActualPos - 5) THEN
		GVL_HMI.bCalHoldSysPressureBt := NOT GVL_IO.gSetSolenoidControl.HoldPressure(); //PressureUp();
	ELSE
		//Raise interlock alarm
		GVL_HMI.bCalHoldSysPressureBt := FALSE;
	END_IF
END_IF

// HMI Button responsible for stopping the leak test
IF GVL_HMI.bCalStopLeakTestBt THEN
	GVL_HMI.bCalStopLeakTestBt := NOT GVL_IO.gSetSolenoidControl.Idle();
END_IF

// Leak test stage Analog input pressure HMI shown
IF GVL_Calibration.eLeakTestState <> E_LeakTestState.IDLE THEN
	GVL_HMI.rCalLeakTestPressure := (GVL_IO.gAnalogInputs.rLeakTestPressureSensor - 220.0) * (3.698 / (6100.0 - 220.0)); // Pressure scaling to PSI
ELSE
	GVL_HMI.rCalLeakTestPressure := 0.00;
END_IF


(* Calibration Procedure *) //---------------------------------------------------------------------------------------------------------------------------------------------

// Calibration procedure trigger
IF GVL_HMI.bStartCalibrationBt THEN

	// Always consume the HMI button request
	GVL_HMI.bStartCalibrationBt := FALSE;

	// Reset start validation feedback
	GVL_Alarms.bInvalidSolventSelection := FALSE;
	GVL_Alarms.sStartCalibrationBlockedReason := '';

	iSelectedSolvent := GVL_HMI.iSelectedCalibrationSolvent;

	// Validate selected solvent number first
	IF (iSelectedSolvent >= 1) AND (iSelectedSolvent <= 4) THEN
		rSelectedSolventDensity := GVL_Settings.stSolventsInfo[iSelectedSolvent].rDensity;
	ELSE
		rSelectedSolventDensity := 0.0;
	END_IF

	// Validate solvent number and density range
	bValidSelectedSolvent :=
		(iSelectedSolvent >= 1) AND
		(iSelectedSolvent <= 4) AND
		(rSelectedSolventDensity > 0.0) AND
		(rSelectedSolventDensity <= 5.0);

	IF bValidSelectedSolvent THEN

		GVL_Calibration.bStartCalibration 	:= TRUE;
		GVL_Calibration.aCalibPumps 		:= GVL_HMI.aCalibPumps;
		GVL_Calibration.iReplicatesSetpoint := GVL_Settings.stCalibParameters.iReplicatesSetpoint;
		GVL_Calibration.rAcceptanceCriteria := GVL_Settings.stCalibParameters.rAcceptanceCriteria;
		GVL_Calibration.iAllowableFailures 	:= GVL_HMI.stHMICalibParameters.iAllowableFailures;
		
		IF GVL_HMI.stHMICalibParameters.bDelayStart THEN
			GVL_Calibration.tDelayStart := DINT_TO_TIME(INT_TO_DINT(GVL_HMI.stHMICalibParameters.iDelayTimeMin) * 1000 * 60 * 60); // hours to ms
		ELSE
			GVL_Calibration.tDelayStart := T#0MS;
		END_IF

		GVL_Calibration.stPumpCalibrationInfo.rSolventDensity := rSelectedSolventDensity;

		// Solvent name - was created as ID but actually is solvent name description
		GVL_Calibration.stPumpCalibrationInfo.iSolventID := GVL_Settings.stSolventsInfo[iSelectedSolvent].sSolventName;

		DB_Create_Calibration.start := TRUE; // Create a new calibration inside the DB.

	ELSE

		// Do not start calibration
		GVL_Calibration.bStartCalibration := FALSE;
		DB_Create_Calibration.start := FALSE;

		GVL_Alarms.bInvalidSolventSelection := TRUE;

		IF (iSelectedSolvent < 1) OR (iSelectedSolvent > 4) THEN
			GVL_Alarms.sStartCalibrationBlockedReason :=
				'Calibration start blocked: selected solvent must be between 1 and 4.';
		ELSIF (rSelectedSolventDensity <= 0.0) OR (rSelectedSolventDensity > 5.0) THEN
			GVL_Alarms.sStartCalibrationBlockedReason :=
				'Calibration start blocked: selected solvent density must be greater than 0 and less than or equal to 5.';
		ELSE
			GVL_Alarms.sStartCalibrationBlockedReason :=
				'Calibration start blocked: invalid solvent selection.';
		END_IF

	END_IF

END_IF

// Calibration procedure calling
fbCalibrationManager(
	bExecute 		:= GVL_Calibration.bStartCalibration,
	rSolventDensity := rSelectedSolventDensity,
	iSolvent 		:= iSelectedSolvent,
	aPumpSettings 	:= GVL_HMI.aCalibPumps,
	tDelayStart 	:= GVL_Calibration.tDelayStart,
	bPrintReport 	:= GVL_Calibration.bPrintWhenComplete,
	aPumpResults 	=> GVL_Calibration.aCalibPumps,
	bDone 			=> GVL_Calibration.bCalibrationDone,
	bBusy 			=> GVL_Calibration.bCalibrationRunning,
	sStatus 		=> GVL_Calibration.sGlobalStatus,
	iDataCount 		=> iDataCount
);

GVL_Calibration.sGlobalStatus := fbCalibrationManager.sStatus;


// Calibration done treatment
IF fbCalibrationManager.bDone THEN

	GVL_Calibration.bStartCalibration := FALSE;
	GVL_Calibration.bStartCreationCalJson := TRUE;

END_IF


// Save calibration report JSON
fbSaveCalReport(
	bExecute          := GVL_Calibration.bStartCreationCalJson,
	sUser             := GVL_Calibration.stPumpCalibrationInfo.iUserID,
	stReportInfo      := GVL_Calibration.stPumpCalReportInfo,
	stCalibrationInfo := GVL_Calibration.stPumpCalibrationInfo,
	aCalibrationData  := GVL_Calibration.stPumpCalibrationData,
	iDataCount        := iDataCount
);


// JSON creation done treatment
IF fbSaveCalReport.bDone THEN

	GVL_Calibration.bCreationCalJsonDone  := TRUE;
	GVL_Calibration.bCreationCalJsonError := FALSE;
	GVL_Calibration.bStartCreationCalJson := FALSE;

	fbCalibrationManager.Reset(bHard := TRUE);
	fbSaveCalReport.Reset();

	GVL_HMI.eMachineMode := E_MachineMode.STOPPED;


// JSON creation error treatment
ELSIF fbSaveCalReport.bError THEN

	GVL_Calibration.bCreationCalJsonDone  := FALSE;
	GVL_Calibration.bCreationCalJsonError := TRUE;

	GVL_Alarms.bCalJsonCreationError := TRUE;
	GVL_Alarms.nCalJsonCreationErrorId := fbSaveCalReport.nErrId;

	fbSaveCalReport.Reset();

END_IF

(* Linear Pumps Enable *) //---------------------------------------------------------------------------------------------------------------------------------------------
IF GVL_HMI.bCalLinearPumpsEnableBt THEN
    // Ensure we have the latest HMI snapshot
    GVL_Calibration.aCalibLinearPumps := GVL_HMI.aCalibLinearPumps;

    IF EnableLinearPumps() THEN
        // Operation finished successfully
        GVL_HMI.bCalLinearPumpsEnableBt := FALSE; // Set Dirty flag that does not allow closing the popup
		GVL_HMI.bCalLinearPumpsDirty := TRUE;
    END_IF
END_IF

(* Linear Pumps Homing *) //---------------------------------------------------------------------------------------------------------------------------------------------
IF GVL_HMI.bCalLinearPumpsHomeBt THEN
    // Ensure we have the latest HMI snapshot
    GVL_Calibration.aCalibLinearPumps := GVL_HMI.aCalibLinearPumps;

    IF HomeLinearPumps() THEN
        GVL_HMI.bCalLinearPumpsHomeBt := FALSE;
		GVL_HMI.bCalLinearPumpsDirty := TRUE; // Set Dirty flag that does not allow closing the popup
    END_IF
END_IF

(* Linear Pumps Moving *) //---------------------------------------------------------------------------------------------------------------------------------------------
IF GVL_HMI.bCalLinearPumpsMoveBt THEN
    // Ensure we have the latest HMI snapshot
    GVL_Calibration.aCalibLinearPumps := GVL_HMI.aCalibLinearPumps;

    IF MoveLinearPumps() THEN
        GVL_HMI.bCalLinearPumpsMoveBt := FALSE;
		GVL_HMI.bCalLinearPumpsDirty := TRUE; // Set Dirty flag that does not allow closing the popup
    END_IF
END_IF

(* Linear Pumps Stop - stops ALL pumps regardless of selection *) // ---------------------------------------------------------------------------------------------------
IF GVL_HMI.bCalLinearPumpsStopBt THEN
    // Immediately requests a "Stop" on every linear pump.
    FOR i := 1 TO 10 DO
        GVL_Motion.aPumpsLinear[i].Stop();
        // Clear any local latches
        aLinearPumpsEnable[i] := FALSE;
        aLinearPumpsHoming[i] := FALSE;
        bLinearPumpsOldPosMove[i] := FALSE;
    END_FOR
    // Reset trigger
    GVL_HMI.bCalLinearPumpsStopBt := FALSE;
END_IF

(* Linear Pumps Save - Gets all new motors position and saves on old position | Disable all pumps that are enabled *)
rtrigSaveLinearPumps(CLK := GVL_HMI.bCalLinearPumpsSaveBt);

IF rtrigSaveLinearPumps.Q THEN
    SaveLinearPumpPositions();
END_IF

(* Valves Manual Movement *) //-----------------------------------------------------------------------------------------------------------------------------------------------------
IF GVL_HMI.bCalMoveValves THEN
	FOR i := 1 TO 5 DO
		IF NOT bMoveValves[i] THEN
			bMoveValves[i] := GVL_Motion.aValvesObj[i].MoveValve( iPosition := GVL_HMI.iCalMoveValvesPosition ,rVelocity := 1500, rAcc := 1000, rDec := 1000);
		END_IF
	END_FOR
END_IF

IF bMoveValves[1] AND bMoveValves[2] AND bMoveValves[3] AND bMoveValves[4] AND bMoveValves[5] THEN
	FOR i := 1 TO 5 DO
			bMoveValves[i] := FALSE;
	END_FOR
	GVL_HMI.bCalMoveValves := FALSE;
END_IF

(* M1 Motor Manual Movement *) //-----------------------------------------------------------------------------------------------------------------------------------------------------
IF GVL_HMI.bCalMoveM1Motor AND GVL_IO.gDigInputs.bThroatJigPresent THEN
	IF NOT bMoveM1Fast THEN
		bMoveM1Fast := GVL_Motion.aMotors[1].MoveAbsolute(	rPosition := GVL_Settings.stMachineParam.aM1Position[GVL_HMI.iCalMoveM1MotorPosition] + GVL_Settings.stMachineParam.fM1PositionDeceleration,
														rVelocity := GVL_Settings.stMachineParam.rM1Velocity,
														rAcc := GVL_Settings.stMachineParam.rM1Accleration,
														rDec := GVL_Settings.stMachineParam.rM1Deceleration
														);
	END_IF
	
	IF bMoveM1Fast AND NOT bMoveM1Slow THEN
		bMoveM1Slow := GVL_Motion.aMotors[1].MoveAbsolute(	rPosition := GVL_Settings.stMachineParam.aM1Position[GVL_HMI.iCalMoveM1MotorPosition],
														rVelocity := GVL_Settings.stMachineParam.rM1PrecisionVelocity,
														rAcc := GVL_Settings.stMachineParam.rM1PrecisionVelocity,
														rDec := GVL_Settings.stMachineParam.rM1PrecisionVelocity
														);
	END_IF
	
	IF bMoveM1Fast AND bMoveM1Slow THEN
		bMoveM1Fast := FALSE;
		bMoveM1Slow := FALSE;
		GVL_HMI.bCalMoveM1Motor := FALSE;
	END_IF									

END_IF

// Temp ## Dosing Test ## -----------------------------------------------

IF bSetDosingPumps THEN
	aDosingPumps[1] := FALSE;
	aDosingPumps[2] := FALSE;
	aDosingPumps[3] := FALSE;
	aDosingPumps[4] := FALSE;
	aDosingPumps[5] := FALSE;
	aDosingPumps[6] := FALSE;
	aDosingPumps[7] := FALSE;
	aDosingPumps[8] := FALSE;
	aDosingPumps[9] := FALSE;
	aDosingPumps[10] := FALSE;
END_IF

IF GVL_Calibration.bDosingTestEnable THEN
	fbDosingTest (	iReplicate := iReplicates,
					bExecute := GVL_Calibration.bDosingTestEnable,
					rVolumeTesting := rTargetVolume,
					aPumps := aDosingPumps
				  );
END_IF

IF fbDosingTest.bDone THEN
	GVL_Calibration.bDosingTestEnable := FALSE;
END_IF

IF bDosingTestReset THEN
	bDosingTestReset := NOT fbDosingTest.Reset();
	bDosingTestReset := FALSE;
END_IF

IF bDosingTestResults THEN
	bDosingTestResults := NOT fbDosingTest.ResetResults();
	bDosingTestResults := FALSE;
END_IF

METHOD EnableLinearPumps : BOOL
VAR_INPUT
END_VAR
VAR
    bAnySelected : BOOL;
    bAllOperational : BOOL;
END_VAR
// Track if at least one pump is selected
bAnySelected := FALSE;
bAllOperational := TRUE;

// Issue enable only for selected pumps
FOR i := 1 TO 10 DO
    IF GVL_Calibration.aCalibLinearPumps[i].bActivate THEN
        bAnySelected := TRUE;
        // Call axis enable if not yet operational
        IF NOT IsAxisOperational(iAxis := i) THEN
            // Fire the enable command to the axis object
            aLinearPumpsEnable[i] := GVL_Motion.aPumpsLinear[i].Enable();
        END_IF
        // After command, check current status
        IF NOT IsAxisOperational(iAxis := i) THEN
            bAllOperational := FALSE; // At least one still not operational
        END_IF
    END_IF
END_FOR

// No selection: nothing to do (fail-safe FALSE)
IF NOT bAnySelected THEN
    EnableLinearPumps := FALSE; // Nothing selected
    RETURN;
END_IF

// Finish when all selected are operational
IF bAllOperational THEN
    // Clear latches
    FOR i := 1 TO 10 DO
        aLinearPumpsEnable[i] := FALSE;
    END_FOR
    EnableLinearPumps := TRUE;
	RETURN;
ELSE
    EnableLinearPumps := FALSE;
END_IF

(*------------------------------------------------------------------------------------------*)
(*
//Enabling Linear Pumps
FOR i := 1 TO 10 DO
	aLinearPumpsEnable[i] := GVL_Motion.aPumpsLinear[i].Enable();
END_FOR

//Testing if all motors were anabled
IF aLinearPumpsEnable[1] AND aLinearPumpsEnable[2] AND aLinearPumpsEnable[3] AND aLinearPumpsEnable[4] AND aLinearPumpsEnable[5] AND aLinearPumpsEnable[6] AND aLinearPumpsEnable[7] AND aLinearPumpsEnable[8] AND aLinearPumpsEnable[9] AND aLinearPumpsEnable[10] THEN
	FOR i := 1 TO 10 DO
		aLinearPumpsEnable[i] := FALSE;
	END_FOR
	EnableLinearPumps := TRUE;
	RETURN;
ELSE
	EnableLinearPumps := FALSE;
END_IF
*)
END_METHOD

METHOD PRIVATE HoldSystemPressure : BOOL
VAR_INPUT
END_VAR
VAR
	bDoneSeen : BOOL := FALSE;
END_VAR
// Queremos: A=TRUE, B=FALSE, C=FALSE
bNeedsSet :=
    (GVL_IO.gDigOutputs.bSolenoidValveA <> TRUE) OR
    (GVL_IO.gDigOutputs.bSolenoidValveB <> FALSE) OR
    (GVL_IO.gDigOutputs.bSolenoidValveC <> FALSE);

IF bNeedsSet THEN
    // Aplica apenas se precisar alterar algo
    GVL_IO.gDigOutputs.bSolenoidValveA := TRUE;
    GVL_IO.gDigOutputs.bSolenoidValveB := FALSE;
    GVL_IO.gDigOutputs.bSolenoidValveC := FALSE;

    // (opcional) limpar flags de outras fases
    bPressureUpSolenoids := FALSE;
    bPressureUpExecute   := FALSE;
	
	GVL_Calibration.eLeakTestState := E_LeakTestState.HOLD_PRESSURE;

    HoldSystemPressure := TRUE;   // retornamos TRUE somente quando houve mudança
ELSE
    HoldSystemPressure := FALSE;  // já estava no estado desejado
END_IF
(*//FB Execute 
fbSolenoidControl( bExecute := bHoldPressureSolenoids, eSolenoidSet := E_SolenoidSet.LEAKTESTMONITORING);

// 0. Trigger
IF NOT bHoldPressureRequested THEN
    bHoldPressureExecute := TRUE;
    bHoldPressureRequested := TRUE;
END_IF

// 1. Close Solenoid B and keep A Open to hold the system pressure
IF bHoldPressureExecute AND bHoldPressureRequested THEN
	bHoldPressureSolenoids := TRUE;
END_IF

IF fbSolenoidControl.bDone THEN
	bDoneSeen := TRUE;
END_IF

// 3. Done - Reset and Return True
IF NOT bHoldPressureSolenoids AND NOT bHoldPressureExecute AND bHoldPressureRequested THEN
	bHoldPressureRequested := FALSE;
	bDoneSeen := FALSE;
	HoldSystemPressure := TRUE;
	RETURN;
ELSE
	HoldSystemPressure := FALSE;
END_IF

// Resetamos o bExecute SOMENTE DEPOIS de ter visto o Done
IF bDoneSeen THEN
	bHoldPressureSolenoids := FALSE;
	bHoldPressureExecute := FALSE;
END_IF*)
END_METHOD

METHOD HomeLinearPumps : BOOL
VAR_INPUT
END_VAR
VAR
	bAnySelected : BOOL;
	bAllHomed : BOOL;
	bAllOldPosMovesDone : BOOL;
	bAllPumpsHomedone : BOOL;
	rPositionTolerance : REAL := 0.05;
END_VAR
bAnySelected := FALSE;
// 1) Trigger homing only for selected & operational axes
FOR i := 1 TO 10 DO
    IF GVL_Calibration.aCalibLinearPumps[i].bActivate THEN
        bAnySelected := TRUE;

        // Interlock: must be Operational before Home
        IF IsAxisOperational(iAxis := i) THEN
            // If not homed yet, keep requesting Home
            IF NOT aLinearPumpsHoming[i] THEN
                aLinearPumpsHoming[i] := GVL_Motion.aPumpsLinear[i].Home(
                    pHomeSensor := ADR(GVL_Motion.aPumps[i].Linear.iHomeSensor.0),
                    rVelocity   := GVL_Motion.aPumps[i].Linear.rHomeVel,
                    rAcc        := GVL_Motion.aPumps[i].Linear.rHomeAcc,
                    rDec        := GVL_Motion.aPumps[i].Linear.rHomeDec
                );
            END_IF
        ELSE
            // Not operational -> cannot home yet
            bAllHomed := FALSE;
        END_IF
	ELSE
		aLinearPumpsHoming[i] := TRUE;
    END_IF
END_FOR

// If none selected, nothing to do
IF NOT bAnySelected THEN
    HomeLinearPumps := FALSE;
    RETURN;
END_IF

// 2) After all selected are homed, move them to OldPosition
bAllHomed := aLinearPumpsHoming[1] AND aLinearPumpsHoming[2] AND aLinearPumpsHoming[3] AND aLinearPumpsHoming[4] AND 
			 aLinearPumpsHoming[5] AND aLinearPumpsHoming[6] AND aLinearPumpsHoming[7] AND aLinearPumpsHoming[8] AND 
			 aLinearPumpsHoming[9] AND aLinearPumpsHoming[10];

IF bAllHomed THEN
    bLinearPumpsOldPosStart := TRUE;
END_IF

// 3) Move to old position only the selected pumps
IF bLinearPumpsOldPosStart THEN
	FOR i := 1 TO 10 DO
		IF GVL_Calibration.aCalibLinearPumps[i].bActivate THEN
			IF NOT bLinearPumpsOldPosMove[i] THEN
				bLinearPumpsOldPosMove[i] := GVL_Motion.aPumpsLinear[i].MoveAbsolute(
					rPosition := GVL_Retain.rLinearPumpOldPosition[i],
					rVelocity := GVL_Motion.aPumps[i].Linear.rHomeVel,
					rAcc      := GVL_Motion.aPumps[i].Linear.rHomeAcc,
					rDec      := GVL_Motion.aPumps[i].Linear.rHomeDec
				);
			END_IF
			IF GVL_Motion.aPumps[i].Linear.rActualPos <= (GVL_Motion.aPumps[i].Linear.rActualPos + rPositionTolerance) AND  GVL_Motion.aPumps[i].Linear.rActualPos >= (GVL_Motion.aPumps[i].Linear.rActualPos - rPositionTolerance) THEN
				bLinearPumpsOldPosMove[i] := TRUE;
			END_IF
		ELSE
			bLinearPumpsOldPosMove[i] := TRUE;
		END_IF
	END_FOR
END_IF

bAllOldPosMovesDone := bLinearPumpsOldPosMove[1] AND bLinearPumpsOldPosMove[2] AND bLinearPumpsOldPosMove[3] AND bLinearPumpsOldPosMove[4] AND bLinearPumpsOldPosMove[5] AND bLinearPumpsOldPosMove[6] AND bLinearPumpsOldPosMove[7] AND bLinearPumpsOldPosMove[8] AND bLinearPumpsOldPosMove[9] AND bLinearPumpsOldPosMove[10];

// 4) Completion and cleanup
IF bAllHomed AND bAllOldPosMovesDone THEN
    FOR i := 1 TO 10 DO
        aLinearPumpsHoming[i] := FALSE;
        bLinearPumpsOldPosMove[i] := FALSE;
    END_FOR
    bLinearPumpsOldPosStart := FALSE;
	bAllHomed	:= FALSE;
	bAllPumpsHomedone := FALSE;
    HomeLinearPumps := TRUE;
	RETURN;
ELSE
    HomeLinearPumps := FALSE;
END_IF
END_METHOD

METHOD IsAxisHomed : BOOL
VAR_INPUT
	iAxis : INT; // axis linear pumps index
END_VAR
// Returns TRUE if axis i is homed in NC
CASE iAxis OF
    1: IsAxisHomed := GVL_HMI.stIOTerm23.bAxisHomed[1]; 
    2: IsAxisHomed := GVL_HMI.stIOTerm24.bAxisHomed[1];
    3: IsAxisHomed := GVL_HMI.stIOTerm25.bAxisHomed[1];
    4: IsAxisHomed := GVL_HMI.stIOTerm26.bAxisHomed[1];
    5: IsAxisHomed := GVL_HMI.stIOTerm27.bAxisHomed[1];
    6: IsAxisHomed := GVL_HMI.stIOTerm28.bAxisHomed[1];
    7: IsAxisHomed := GVL_HMI.stIOTerm29.bAxisHomed[1];
    8: IsAxisHomed := GVL_HMI.stIOTerm30.bAxisHomed[1];
    9: IsAxisHomed := GVL_HMI.stIOTerm31.bAxisHomed[1];
    10: IsAxisHomed := GVL_HMI.stIOTerm32.bAxisHomed[1];
ELSE
    IsAxisHomed := FALSE;
END_CASE
END_METHOD

METHOD IsAxisOperational : BOOL
VAR_INPUT
	iAxis : INT; // axis linear pumps index
END_VAR
// Returns TRUE if axis i is operational (enabled) in NC
CASE iAxis OF
    1: IsAxisOperational := GVL_HMI.stIOTerm23.bAxisOperational[1]; 
    2: IsAxisOperational := GVL_HMI.stIOTerm24.bAxisOperational[1];
    3: IsAxisOperational := GVL_HMI.stIOTerm25.bAxisOperational[1];
    4: IsAxisOperational := GVL_HMI.stIOTerm26.bAxisOperational[1];
    5: IsAxisOperational := GVL_HMI.stIOTerm27.bAxisOperational[1];
    6: IsAxisOperational := GVL_HMI.stIOTerm28.bAxisOperational[1];
    7: IsAxisOperational := GVL_HMI.stIOTerm29.bAxisOperational[1];
    8: IsAxisOperational := GVL_HMI.stIOTerm30.bAxisOperational[1];
    9: IsAxisOperational := GVL_HMI.stIOTerm31.bAxisOperational[1];
    10: IsAxisOperational := GVL_HMI.stIOTerm32.bAxisOperational[1];
ELSE
    IsAxisOperational := FALSE;
END_CASE
END_METHOD

METHOD MoveLinearPumps : BOOL
VAR_INPUT
END_VAR
VAR
	bAnySelected : BOOL;
    bAllMovesDone : BOOL;
END_VAR
bAnySelected := FALSE;

FOR i := 1 TO 10 DO
    IF GVL_Calibration.aCalibLinearPumps[i].bActivate THEN
        bAnySelected := TRUE;

        // Interlocks: must be Operational and Homed before move
        IF IsAxisOperational(iAxis := i) AND IsAxisHomed(iAxis := i) THEN
            // Issue move if not already "in progress/done" (implement your latch if needed)
            // We'll reuse bLinearPumpsOldPosMove[] as generic "move latch"
            IF NOT bLinearPumpsOldPosMove[i] THEN
                bLinearPumpsOldPosMove[i] := GVL_Motion.aPumpsLinear[i].MoveAbsolute(
                    rPosition := GVL_Calibration.aCalibLinearPumps[i].rNewPosition,
                    rVelocity := GVL_Motion.aPumps[i].Linear.rHomeVel,
                    rAcc      := GVL_Motion.aPumps[i].Linear.rHomeAcc,
                    rDec      := GVL_Motion.aPumps[i].Linear.rHomeDec
                );
            END_IF
        ELSE
            // Interlock not satisfied -> cannot move
            bAllMovesDone := FALSE;
        END_IF
	ELSE
		bLinearPumpsOldPosMove[i] := TRUE;
    END_IF
END_FOR

IF NOT bAnySelected THEN
    MoveLinearPumps := FALSE; // nothing selected
    RETURN;
END_IF

bAllMovesDone := bLinearPumpsOldPosMove[1] AND bLinearPumpsOldPosMove[2] AND bLinearPumpsOldPosMove[3] AND 
				 bLinearPumpsOldPosMove[4] AND bLinearPumpsOldPosMove[5] AND bLinearPumpsOldPosMove[6] AND 
				 bLinearPumpsOldPosMove[7] AND bLinearPumpsOldPosMove[8] AND bLinearPumpsOldPosMove[9] AND 
				 bLinearPumpsOldPosMove[10];

IF bAllMovesDone THEN
    // Clear latches for next command
    FOR i := 1 TO 10 DO
        bLinearPumpsOldPosMove[i] := FALSE;
    END_FOR
	bAllMovesDone := FALSE;
	bAnySelected := FALSE;
    MoveLinearPumps := TRUE;
	RETURN;
ELSE
    MoveLinearPumps := FALSE;
END_IF
END_METHOD

METHOD PRIVATE PressureUp : BOOL
VAR_INPUT
END_VAR
VAR
	bDoneSeen : BOOL := FALSE;
	bPressureDone : BOOL := FALSE;
END_VAR
// Saída padrão
PressureUp := FALSE;

// --- FSM ---
CASE ePState OF

    E_PState.Init:
        // Disparo único por chamada (se quiser condicionar, coloque aqui um bExecute)
        bMoveIssued := FALSE;
        tonSealTimeout(IN := FALSE);
        ePState := E_PState.SealIssue;

    E_PState.SealIssue:
        // Interlock: sem jig, não segue
        IF NOT GVL_IO.gDigInputs.bThroatJigPresent THEN
            GVL_HMI.bM1MoveNotAllowedTrigger := TRUE;  // opcional: gatilho de alarme
            ePState := E_PState.Fault;
        ELSE
            // Emite o comando uma única vez
            bMoveIssued := GVL_Motion.aMotors[1].MoveAbsolute(
                rPosition := GVL_Settings.stMachineParam.aM1Position[2],   // Seal pos
                rVelocity := GVL_Settings.stMachineParam.rM1Velocity,
                rAcc      := GVL_Settings.stMachineParam.rM1Accleration,
                rDec      := GVL_Settings.stMachineParam.rM1Deceleration
            );
            tonSealTimeout(IN := TRUE, PT := T#10S);
            ePState := E_PState.SealWait;
        END_IF

    E_PState.SealWait:
        // Aguarda o Done do movimento
        IF GVL_Motion.aMotors[1].MoveAbsolute(
            rPosition := GVL_Settings.stMachineParam.aM1Position[2],
            rVelocity := GVL_Settings.stMachineParam.rM1Velocity,
            rAcc      := GVL_Settings.stMachineParam.rM1Accleration,
            rDec      := GVL_Settings.stMachineParam.rM1Deceleration
        ) THEN
            tonSealTimeout(IN := FALSE);
            ePState := E_PState.OpenValves;
        ELSE
            // Timeout de segurança
            tonSealTimeout(IN := TRUE);
            IF tonSealTimeout.Q THEN
                ePState := E_PState.Fault;
            END_IF
        END_IF

    E_PState.OpenValves:
        // Pressuriza o sistema: A/B abertas, C fechada
        IF GVL_IO.gSetSolenoidControl.PressureUp() THEN
			ePState := E_PState.Done;
		END_IF

    E_PState.Done:
		GVL_Calibration.eLeakTestState := E_LeakTestState.PRESSURE_UP;
        bMoveIssued := FALSE;
        tonSealTimeout(IN := FALSE);
		PressureUp := TRUE;          // pulso de sucesso nesta chamada
        ePState := E_PState.Init;    // pronto para próximo ciclo
        RETURN;                      // encerra o método neste ciclo

    E_PState.Fault:
        // Falha: garanta estado seguro (não pressuriza)
        (*GVL_IO.gDigOutputs.bSolenoidValveA := FALSE;
        GVL_IO.gDigOutputs.bSolenoidValveB := FALSE;
        GVL_IO.gDigOutputs.bSolenoidValveC := FALSE;*)
		GVL_IO.gSetSolenoidControl.Idle();
        bMoveIssued := FALSE;
        tonSealTimeout(IN := FALSE);
        PressureUp := FALSE;
        ePState := E_PState.Init;             // ou mantenha em Fault até um reset externo
        RETURN;

ELSE
    // Recuperação defensiva
    ePState := E_PState.Init;
END_CASE

(*//FB Execute 
fbSolenoidControl( bExecute := bPressureUpSolenoids, eSolenoidSet := E_SolenoidSet.LEAKTEST);

// 0. Trigger
IF NOT bPressureUpRequested THEN
    bPressureUpExecute := TRUE;
	bSealStages	:= TRUE;
    bPressureUpRequested := TRUE;
END_IF

// 1. Sealing Stages (M1 axis)
IF bSealStages THEN
	bSealStages := NOT GVL_Motion.aMotors[1].MoveAbsolute( rPosition := GVL_Settings.stMachineParam.aM1Position[2], rVelocity := GVL_Settings.stMachineParam.rM1Velocity, rAcc := GVL_Settings.stMachineParam.rM1Accleration, rDec := GVL_Settings.stMachineParam.rM1Deceleration);
END_IF

// 2. Open Solenoid B and A to pressure up the system
IF NOT bSealStages AND bPressureUpRequested THEN
	bPressureUpSolenoids := TRUE;
END_IF

IF fbSolenoidControl.bDone THEN
	bDoneSeen := TRUE;
END_IF

// 3. Done - Reset and Return True
IF bPressureUpRequested AND NOT bPressureUpExecute AND NOT bSealStages THEN
	bPressureUpRequested := FALSE;
	bDoneSeen	:= FALSE;
	PressureUp 	:= TRUE;
	RETURN;
ELSE
	PressureUp := FALSE;
END_IF

// Resetamos o bExecute SOMENTE DEPOIS de ter visto o Done
IF bDoneSeen THEN
	bPressureUpSolenoids := FALSE;
	bPressureUpExecute := FALSE;
END_IF

*)
END_METHOD

METHOD Reset : BOOL
VAR_INPUT
END_VAR
Reset := FALSE;

// 1) First entry: clear everything ONCE
IF NOT bResetRequested THEN
    bResetRequested := TRUE;

    // Reset Calibration Flags (tudo o que você já limpa hoje)
    bLeakTestReset := FALSE;

    bStartCalibrationPrev := FALSE;
    bStartCalibrationEdge := FALSE;

    bLinearPumpsEnabled      := FALSE;
    bLinearPumpsHomed        := FALSE;
    bLinearPumpsOldPosStart  := FALSE;
    bLinearPumpsOldPosDone   := FALSE;

    eStopState := E_StopState.Init;
    ePState    := E_PState.Init;
    GVL_Calibration.eLeakTestState := E_LeakTestState.IDLE;

    bPressureUpExecute      := FALSE;
    bPressureUpRequested    := FALSE;
    bSealStages             := FALSE;
    bPressureUpSolenoids    := FALSE;
    bHoldPressureExecute    := FALSE;
    bHoldPressureRequested  := FALSE;
    bHoldPressureSolenoids  := FALSE;
    bStopLeakTestExecute    := FALSE;
    bStopLeakTestRequested  := FALSE;
    bStopLeakTestSolenoids  := FALSE;

    bMoveIssued := FALSE;
    bNeedsSet   := FALSE;

    tonSealTimeout(IN := FALSE);
    tonResetMotorDelay(IN := FALSE);

    bStopM1Motor  := FALSE;
    bResetM1Motor := FALSE;
	
	GVL_Calibration.sGlobalStatus := 'Idle';

    // arrays / buffers
    FOR i := 1 TO 5 DO
        bMoveValves[i] := FALSE;
    END_FOR

    FOR i := 1 TO 10 DO
        aLinearPumpsEnable[i]      := FALSE;
        aLinearPumpsHoming[i]      := FALSE;
        bLinearPumpsOldPosMove[i]  := FALSE;
        aLinearPumpsMoveDone[i]    := FALSE;
    END_FOR

    FOR i := 1 TO 100 DO
        GVL_Calibration.stPumpCalibrationData[i].dDateTime := '';
        GVL_Calibration.stPumpCalibrationData[i].iPumpNumber := 0;
        GVL_Calibration.stPumpCalibrationData[i].iPumpRevs := 0;
        GVL_Calibration.stPumpCalibrationData[i].rCriteria := 0.0;
        GVL_Calibration.stPumpCalibrationData[i].rDifferencePercent := 0.0;
        GVL_Calibration.stPumpCalibrationData[i].rDifferenceUl := 0.0;
        GVL_Calibration.stPumpCalibrationData[i].rGrossWeigth := 0.0;
        GVL_Calibration.stPumpCalibrationData[i].rNetVolume := 0.0;
        GVL_Calibration.stPumpCalibrationData[i].rNetWeigth := 0.0;
        GVL_Calibration.stPumpCalibrationData[i].rTareWeigth := 0.0;
        GVL_Calibration.stPumpCalibrationData[i].rTargetVolume := 0.0;
        GVL_Calibration.stPumpCalibrationData[i].sStep := '';
    END_FOR
	
	fbSaveCalReport.Reset();

    // IMPORTANT: Resets bResetDone here (1x)
    bResetDone := FALSE;
END_IF

// 2) Run the manager reset until done
IF NOT bResetDone THEN
    bResetDone := fbCalibrationManager.Reset(bHard := TRUE);
END_IF

// 3) Finish (one pulse)
IF bResetDone THEN
    bResetRequested := FALSE;
    bResetDone := FALSE; 
    Reset := TRUE;
    RETURN;
END_IF

(*
//Reset Calibration Flags
bLeakTestReset := FALSE;
bResetDone := FALSE;

bStartCalibrationPrev := FALSE;
bStartCalibrationEdge := FALSE;

bLinearPumpsEnabled		 := FALSE;
bLinearPumpsHomed		 := FALSE;
bLinearPumpsOldPosStart	 := FALSE;
bLinearPumpsOldPosDone	 := FALSE;

eStopState 	 	:= E_StopState.Init;
ePState 		:= E_PState.Init;	
GVL_Calibration.eLeakTestState 	:= E_LeakTestState.IDLE;

bPressureUpExecute 		 := FALSE;
bPressureUpRequested 	 := FALSE;
bSealStages				 := FALSE;
bPressureUpSolenoids	 := FALSE;
bHoldPressureExecute 	 := FALSE;
bHoldPressureRequested 	 := FALSE;
bHoldPressureSolenoids	 := FALSE;
bStopLeakTestExecute 	 := FALSE;
bStopLeakTestRequested 	 := FALSE;
bStopLeakTestSolenoids 	 := FALSE;

bMoveIssued      := FALSE;
bNeedsSet 		 := FALSE;

tonSealTimeout(IN := FALSE);
tonResetMotorDelay(IN := FALSE);

bStopM1Motor 			 := FALSE;
bResetM1Motor 			 := FALSE;


bLinearPumpsEnabled		 := FALSE;
bLinearPumpsHomed		 := FALSE;
bLinearPumpsOldPosStart	 := FALSE;
bLinearPumpsOldPosDone	 := FALSE;
bLinearPumpsMove		 := FALSE;

bCalPressureUpSystemBt	 := FALSE;

FOR i := 1 TO 5 DO
	bMoveValves[i] := FALSE;
END_FOR

FOR i := 1 TO 10 DO
	aLinearPumpsEnable[i] := FALSE;
	aLinearPumpsHoming[i] := FALSE;
	bLinearPumpsOldPosMove[i] := FALSE;
	aLinearPumpsMoveDone[i] := FALSE;
END_FOR

FOR i := 1 TO 100 DO
	GVL_Calibration.stPumpCalibrationData[i].dDateTime 			:= '';
	GVL_Calibration.stPumpCalibrationData[i].iPumpNumber 		:= 0;
	GVL_Calibration.stPumpCalibrationData[i].iPumpRevs 			:= 0;
	GVL_Calibration.stPumpCalibrationData[i].rCriteria 			:= 0.0;
	GVL_Calibration.stPumpCalibrationData[i].rDifferencePercent := 0.0;
	GVL_Calibration.stPumpCalibrationData[i].rDifferenceUl 		:= 0.0;
	GVL_Calibration.stPumpCalibrationData[i].rGrossWeigth 		:= 0.0;
	GVL_Calibration.stPumpCalibrationData[i].rNetVolume 		:= 0.0;
	GVL_Calibration.stPumpCalibrationData[i].rNetWeigth 		:= 0.0;
	GVL_Calibration.stPumpCalibrationData[i].rTareWeigth 		:= 0.0;
	GVL_Calibration.stPumpCalibrationData[i].rTargetVolume 		:= 0.0;
	GVL_Calibration.stPumpCalibrationData[i].sStep 				:= '';
END_FOR

IF NOT bResetDone THEN
	bResetDone := fbCalibrationManager.Reset(bHard := TRUE);
ELSE
	Reset := TRUE;
	RETURN;
END_IF
*)
END_METHOD

METHOD SaveLinearPumpPositions : BOOL
VAR
	i               : INT;
    bAnyChange      : BOOL := FALSE;
    bDisableDone    : BOOL;
    rSavedPos       : LREAL;
    rActualPos      : LREAL;
    lrTolerance     : LREAL := 2;
END_VAR
bAnyChange := FALSE;

FOR i := 1 TO 10 DO

    // Default metadata for all records
    GVL_Calibration.stLinearCalibrationData[i].sPumpNumber   := TO_STRING(i);
    GVL_Calibration.stLinearCalibrationData[i].sUserName     := GVL_HMI.sUserNameEventTriggered;
    GVL_Calibration.stLinearCalibrationData[i].sDateOfChange := GVL_HMI.sDateAndTimeEventTriggered;

    rSavedPos  := GVL_Retain.rLinearPumpOldPosition[i];
    rActualPos := GVL_Motion.aPumps[i].Linear.rActualPos;

    // Only trust actual position if axis is enabled + homed
    IF GVL_Motion.aPumps[i].Linear.iOperational AND GVL_Motion.aPumps[i].Linear.iHomed THEN

        // Compare saved vs actual to decide if there was a real position change
        IF ABS(rActualPos - rSavedPos) > lrTolerance THEN

            // Fill DB payload
            GVL_Calibration.stLinearCalibrationData[i].sOldPosition := TO_STRING(rSavedPos);
            GVL_Calibration.stLinearCalibrationData[i].sNewPosition := TO_STRING(rActualPos);

			// Update HMI Values
			GVL_HMI.aCalibLinearPumps[i].rOldPosition := rSavedPos;
			GVL_HMI.aCalibLinearPumps[i].rNewPosition := rActualPos;
			
            // Update local retained reference
            GVL_Retain.rLinearPumpOldPosition[i] := rActualPos;

            bAnyChange := TRUE;

        ELSE
            // No real change
            GVL_Calibration.stLinearCalibrationData[i].sOldPosition := TO_STRING(rSavedPos);
            GVL_Calibration.stLinearCalibrationData[i].sNewPosition := TO_STRING(rSavedPos);
        END_IF

        // Disable axis after save check
        bDisableDone := GVL_Motion.aPumpsLinear[i].Disable();

    ELSE
        // Axis not valid -> do not trust actual position, do not overwrite retain
        GVL_Calibration.stLinearCalibrationData[i].sOldPosition := TO_STRING(rSavedPos);
        GVL_Calibration.stLinearCalibrationData[i].sNewPosition := TO_STRING(rSavedPos);
    END_IF

END_FOR

// Trigger DB only if at least one pump actually changed
IF bAnyChange THEN
    DB_Query.state := E_DB_QUERY_STATE.INSERT_LINEAR_MOTORS;
END_IF

// Final housekeeping
GVL_HMI.bCalLinearPumpsSaveBt := FALSE;		// Resets the button trigger 
GVL_HMI.bCalLinearPumpsDirty := TRUE;		// Resets the Dirty flag that allow the popup closes
GVL_HMI.sUserNameEventTriggered := '';		// Resets Username triggered from HMI
GVL_HMI.sDateAndTimeEventTriggered := '';	// Resets Date and Time trigerred from HMI
END_METHOD

METHOD PRIVATE StopLeakTest : BOOL
VAR_INPUT
END_VAR
VAR
	bDoneSeen : BOOL := FALSE;
	bMoveM1HomePos : BOOL := FALSE;
	bMotorMoving : BOOL := FALSE;
END_VAR
CASE eStopState OF
    E_StopState.Init:
		StopLeakTest := FALSE;
        bStopLeakTestRequested := TRUE;
		tonResetMotorDelay(IN := FALSE); 
        eStopState := E_StopState.StopMotor;

    E_StopState.StopMotor:
        IF GVL_Motion.aMotors[1].Stop() THEN
            eStopState := E_StopState.CloseSolenoids;
        END_IF

    E_StopState.CloseSolenoids:
        GVL_IO.gDigOutputs.bSolenoidValveA := FALSE;
        GVL_IO.gDigOutputs.bSolenoidValveB := FALSE;
        GVL_IO.gDigOutputs.bSolenoidValveC := FALSE;
        tonResetMotorDelay(IN := TRUE, PT := T#1S);
        eStopState := E_StopState.Delay;

    E_StopState.Delay:
        tonResetMotorDelay(IN := TRUE);
        IF tonResetMotorDelay.Q THEN
            tonResetMotorDelay(IN := FALSE);
            eStopState := E_StopState.ResetMotor;
        END_IF

    E_StopState.ResetMotor:
        IF GVL_Motion.aMotors[1].Reset() THEN
            eStopState := E_StopState.MoveHome;
        END_IF

    E_StopState.MoveHome:
        IF GVL_Motion.aMotors[1].MoveAbsolute(
            rPosition := GVL_Settings.stMachineParam.aM1Position[1],
            rVelocity := GVL_Settings.stMachineParam.rM1Velocity,
            rAcc      := GVL_Settings.stMachineParam.rM1Accleration,
            rDec      := GVL_Settings.stMachineParam.rM1Deceleration) THEN
            eStopState := E_StopState.Done;
        END_IF

    E_StopState.Done:
		GVL_Calibration.eLeakTestState := E_LeakTestState.IDLE;
		bStopLeakTestRequested := FALSE;
        StopLeakTest         := TRUE;
        eStopState := E_StopState.Init; // ou manter em Done até novo comando
		RETURN;
END_CASE

(*// FB Execute 
fbSolenoidControl( bExecute := bStopLeakTestSolenoids, eSolenoidSet := E_SolenoidSet.IDLE);

//Timer Delay between stop and reset the motor
IF bStopM1Motor AND bStopLeakTestSolenoids THEN
	tonResetMotorDelay(in := TRUE, pt := T#1S);
ELSE
	tonResetMotorDelay(in := FALSE, pt := T#1S);
END_IF

// CLean Internal flags
GVL_HMI.bCalPressureUpSystemBt := FALSE;
GVL_HMI.bCalHoldSysPressureBt := FALSE;

// 0. Trigger
IF NOT bStopLeakTestRequested THEN
    bStopLeakTestExecute := TRUE;
    bStopLeakTestRequested := TRUE;
END_IF

// 1. Stop Motor M1
IF NOT bStopM1Motor THEN
	bStopM1Motor := GVL_Motion.aMotors[1].Stop();
END_IF

// 2. Close Solenoid B and C 
IF bStopM1Motor AND NOT bStopLeakTestExecute AND bStopLeakTestRequested THEN
	bStopLeakTestSolenoids := TRUE;
END_IF

IF fbSolenoidControl.bDone THEN
	bDoneSeen := TRUE;
END_IF

// 3. Reset Motor M1
IF tonResetMotorDelay.Q AND NOT bResetM1Motor THEN
	bResetM1Motor := GVL_Motion.aMotors[1].Reset();
END_IF

// 4. Done - Reset and Return True
IF NOT bStopLeakTestSolenoids AND NOT bStopLeakTestExecute AND bStopLeakTestRequested AND bResetM1Motor THEN
	bStopM1Motor := FALSE;
	bResetM1Motor := FALSE;
	bStopLeakTestRequested := FALSE;
	tonResetMotorDelay(in := FALSE);
	bDoneSeen := TRUE;
	StopLeakTest := TRUE;
	RETURN;
ELSE
	StopLeakTest := FALSE;
END_IF

// Resetamos o bExecute SOMENTE DEPOIS de ter visto o Done
IF bDoneSeen THEN
	bStopLeakTestSolenoids := FALSE;
	bStopLeakTestExecute := FALSE;
END_IF*)
END_METHOD

END_PROGRAM

// ---- POUs/5. Calibration/FB_CalibrationManager.TcPOU
FUNCTION_BLOCK FB_CalibrationManager
VAR_INPUT
    bExecute         : BOOL; // Trigger to start calibration
    iSolvent         : USINT; // Selected solvent type
	rSolventDensity  : LREAL; //Solvent Density
    aPumpSettings    : ARRAY[1..10] OF ST_CalibrationPump; // Pump input settings
    tDelayStart      : TIME; // Optional delay before calibration starts
    bPrintReport     : BOOL; // Option to print report at end
END_VAR

VAR_OUTPUT
    aPumpResults     : ARRAY[1..10] OF ST_CalibrationPump; // Pump result structure
    bDone            : BOOL; // Signals end of calibration
    bBusy            : BOOL; // Calibration in progress
    sStatus          : STRING; // Textual status
	iDataCount		 : INT; // Number of positions used into GVL_Calibration.aCalibCheckResult array
END_VAR

VAR
    eStep             	  : E_CalibStep := E_CalibStep.IDLE; // Main step enum
    iPumpIndex        	  : UINT := 1; // Tracks current pump
    iReplicate        	  : UINT := 0; // Tracks current replicate
	bStartCalibration 	  : BOOL := FALSE;
	bCalibrationRequested : BOOL := FALSE;

    tonCalDelay      : TON; // General delay timer
    tonStepTimeout   : TON; // Timeout per step
	tonMotorsDelay	 : TON; // Delay time after positioning the motors
	tonAirDry		 : TON; // Timer to be using air if needed after calibration
	tonWeigthStabilization : TON; //Time after the pump finish to wait for stable weigth
	
	bExecutePulse   : R_TRIG; // Edge detection for bExecute

    aPumpMask        : ARRAY[1..10] OF BOOL; // Mask for pump selection
    aVolumeSetpoint  : ARRAY[1..10] OF REAL; // Target volume for each pump
    aDirection       : ARRAY[1..10] OF E_PumpDirection; // Direction per pump
    aVelocity        : ARRAY[1..10] OF REAL; // Velocity per pump

    fbPumps          	: FB_AllPumpsController; // Instance of pump controller
    rWeightBefore    	: LREAL; // Weight before pump operation
    rWeightAfter     	: LREAL; // Weight after pump operation
    rWeightDelta     	: LREAL; // Weight difference
	rVolume			 	: LREAL; // Volume calculated
	rPumpVolumeSum	 	: LREAL := 0.00; // Sum volume for each pump for average calculus
	rTareWeightSum		: LREAL := 0.00; // Sum Tare Weigth for each pump for average calculus
	rGrossWeightSum		: LREAL := 0.00; // Sum Gross Weigth for each pump for average calculus
	rPumpAverageVolume 	: LREAL := 0.00; // Calculated average volume of each pump at the end of replicates 
	rPumpAvgTareWeigth 	: LREAL := 0.00; // Calculated average Tare Weitgh of each pump at the end of replicates 
	rPumpAvgGrossWeigth	: LREAL := 0.00; // Calculated average Gross Weigth of each pump at the end of replicates 
    bRequestWeight   	: BOOL := FALSE; // Trigger for requesting scale
	bWeightReady	 	: BOOL := FALSE; // Trigger when weigth is ready
	bPumpAdjustNeed	 	: BOOL := FALSE; // Flag that indicates if the checking pump needs to be adjusted or not. 
	bAirDryTrigger		: BOOL := FALSE; // Flag to trigger the air dry timer. 
    rScaleWeight     	: LREAL; // Latest scale result
	rDistanceByVol	 	: LREAL; // MoveRelative distance
	rPercentDifference 	: LREAL; // Percentual Difference between net volume and tagert volume
	iNumberOfAdjusts	: UINT;  // Count of adjustments needed for each pump index
	rPosTolerance		: LREAL := 5.0; // Position Tolerance in mm to make sure there is no noise in the reading
	rFillJarTotalVol 	: LREAL;
	rEmptyJarTotalVol	: LREAL;
	
    rAcceptanceCrit  : REAL := 0.5; // Acceptance percentage (from HMI)
    iAllowableFail   : INT := 2; 	// Max failures from pump settings
    iMaxReplicates   : INT := 2; 	// Replicate count (from HMI)
	iResultIndex	 : INT;	// Array index on calibration results
	
	bMovePump		 : BOOL := FALSE;
	bMoveMotorM1     : BOOL := FALSE; // Motion trigger M1
    bMoveMotorM2     : BOOL := FALSE; // Motion trigger M2
    bMoveMotorM3     : BOOL := FALSE; // Motion trigger M3
	bSetSolenoids	 : BOOL := FALSE; // SetSolenoids flag
    bMoveValve       : ARRAY[1..5] OF BOOL; // Valve position tracking
	bDataBaseSeq	 : BOOL := FALSE;
	

    i                : USINT;// Loop index helper
    bBoxPresent      : BOOL; // True if calibration box detected
    bBoxWeightOK     : BOOL; // True if calibration box has valid weight

    tStepTimeout     : TIME := T#60S; // Default timeout per step;
	tWeightStable	 : TIME := T#10S; // Default waiting time befe request weight
	
	bScalePlausible : BOOL := FALSE; // Plausibility window flag
    bScaleInvalid   : BOOL := FALSE; // Invalid scale response flag
	
	// Scale-attention handling (9999 pause)
    bScaleAttention  : BOOL := FALSE; // TRUE while waiting operator
	bCalBoxAttention : BOOL := FALSE; // TRUE while waiting operator
    eStepResume      : E_CalibStep := E_CalibStep.IDLE; // Step to return to after fix
	
	// Timestamp generation (local system time)
    fbLocalSystemTime : FB_LocalSystemTime;
    stLocal           : TIMESTRUCT;
    sStamp            : STRING(32);
    sHH               : STRING(2);
    sMM               : STRING(2);
    sSS               : STRING(2);
    sMMo              : STRING(3);
    sDD               : STRING(2);
	bDTReady		  : BOOL := FALSE;
	
	//LoadBar UI
	tonProgress : TON;
    sPrev       : STRING(120);
    tPT         : TIME;

    // helpers time calc (seconds)
    rDeltaM2, rDeltaM3, rVM2, rVM3  : LREAL;
    rPumpVelDeg, rRunVelDeg         : LREAL;
    rSecs  							: LREAL;
	
END_VAR

// bExecute Rising edge
bExecutePulse(CLK := bExecute);

// FB Trigger
IF bExecutePulse.Q AND eStep = E_CalibStep.IDLE THEN
    bStartCalibration := TRUE;
END_IF

// Abort logic
IF GVL_HMI.bAbortCalibrationBT THEN
    eStep := E_CalibStep.ERROR;
END_IF

// State machine
CASE eStep OF

    E_CalibStep.IDLE:
    	bBusy := FALSE;
		bDone := FALSE;
		sStatus := 'Idle';
		IF bStartCalibration THEN
			bBusy := TRUE;
			ACT_CleanStart();
			eStep := E_CalibStep.DELAY;
		END_IF

    E_CalibStep.DELAY:

        tonCalDelay(IN := TRUE, PT := tDelayStart);
        sStatus := 'Waiting delay...';
        IF tonCalDelay.Q THEN
            tonCalDelay(IN := FALSE);
            tonStepTimeout(IN := FALSE);
            eStep := E_CalibStep.CHECKING_WEIGH;
			bRequestWeight := TRUE;
			bBoxWeightOK := FALSE;
			bWeightReady := FALSE;
        END_IF

	
    E_CalibStep.CHECKING_WEIGH:
		// ----------------------------------------------------
		// Step guards / status
		// ----------------------------------------------------
		tonStepTimeout(IN := TRUE, PT := tStepTimeout);
		sStatus := 'Checking the Calibration Box Weigth';
	
		bBoxPresent := GVL_IO.gDigInputs.bCalibrationBoxPresent;
	
		// ----------------------------------------------------
		// 1) Global guards first (avoid processing stale values)
		// ----------------------------------------------------
		IF tonStepTimeout.Q THEN
			sStatus := 'Timeout while checking scale';
			eStep := E_CalibStep.ERROR;
	
		ELSIF NOT bBoxPresent THEN
			sStatus := 'Calibration box not present!';
	
			// Defensive cleanup (avoid sticky UI flags)
			GVL_HMI.bCalBoxNeedsAttention := FALSE;
			bCalBoxAttention := FALSE;
	
			// Clear local request state
			bRequestWeight := FALSE;
	
			eStep := E_CalibStep.IDLE;
	
		ELSE
			// ----------------------------------------------------
			// 2) Request weight (non-blocking)
			// ----------------------------------------------------
			IF bRequestWeight THEN
				// This returns the "current" weight value (may be old until ready)
				rScaleWeight := GVL_Calibration.fbScaleDevice.RequestWeight();
	
				// ------------------------------------------------
				// 3) Process only when the device says it's ready
				//    (treat bWeightReady as an event)
				// ------------------------------------------------
				IF GVL_Calibration.fbScaleDevice.bWeightReady THEN
	
					// ---- scale response plausibility window
					bScalePlausible := (rScaleWeight > 0.0) AND (rScaleWeight < 1215.0);
					bScaleInvalid   := (rScaleWeight = 9999.0) OR (NOT bScalePlausible);
	
					// ------------------------------------------------
					// 3a) Scale invalid -> SCALE_ATTENTION (priority)
					// ------------------------------------------------
					IF bScaleInvalid THEN
						tonCalDelay(IN := FALSE);
						tonStepTimeout(IN := FALSE);
						tonWeigthStabilization(IN := FALSE);
	
						// Prevent cascade: if scale is faulty, do not allow CalBox popup to stack behind
						GVL_HMI.bCalBoxNeedsAttention := FALSE;
						bCalBoxAttention := FALSE;
	
						GVL_HMI.bScaleNeedsAtention := TRUE;
						bScaleAttention := TRUE;
	
						// Stop requesting until operator continues
						bRequestWeight := FALSE;
	
						eStepResume := E_CalibStep.CHECKING_WEIGH;
						eStep := E_CalibStep.SCALE_ATTENTION;
	
					ELSE
						// ------------------------------------------------
						// 3b) Scale valid -> evaluate box weight range
						// ------------------------------------------------
						bBoxWeightOK := (rScaleWeight >= 1100.0) AND (rScaleWeight <= 1300.0);
	
						IF NOT bBoxWeightOK THEN
							tonCalDelay(IN := FALSE);
							tonStepTimeout(IN := FALSE);
							tonWeigthStabilization(IN := FALSE);
	
